   1:  PR[91,1] = PR[90,1] + -17.467;
   1:  PR[91,2] = PR[90,2] + 18.172;
   1:  PR[91,3] = PR[90,3] + 44.691;
   1:L PR[91] R[100]mm/sec CNT100;
   1:  PR[91,1] = PR[90,1] + -18.396;
   1:  PR[91,2] = PR[90,2] + 17.648;
   1:  PR[91,3] = PR[90,3] + 44.700;
   1:L PR[91] R[100]mm/sec CNT100;
   1:  PR[91,1] = PR[90,1] + -19.296;
   1:  PR[91,2] = PR[90,2] + 17.079;
   1:  PR[91,3] = PR[90,3] + 44.709;
   1:L PR[91] R[100]mm/sec CNT100;
   1:  PR[91,1] = PR[90,1] + -19.802;
   1:  PR[91,2] = PR[90,2] + 16.724;
   1:  PR[91,3] = PR[90,3] + 44.717;
   1:L PR[91] R[100]mm/sec CNT100;
   1:  PR[91,1] = PR[90,1] + -20.163;
   1:  PR[91,2] = PR[90,2] + 16.469;
   1:  PR[91,3] = PR[90,3] + 44.723;
   1:L PR[91] R[100]mm/sec CNT100;
   1:  PR[91,1] = PR[90,1] + -20.998;
   1:  PR[91,2] = PR[90,2] + 15.816;
   1:  PR[91,3] = PR[90,3] + 44.726;
   1:L PR[91] R[100]mm/sec CNT100;
   1:  PR[91,1] = PR[90,1] + -21.796;
   1:  PR[91,2] = PR[90,2] + 15.125;
   1:  PR[91,3] = PR[90,3] + 44.735;
   1:L PR[91] R[100]mm/sec CNT100;
   1:  PR[91,1] = PR[90,1] + -22.555;
   1:  PR[91,2] = PR[90,2] + 14.396;
   1:  PR[91,3] = PR[90,3] + 44.744;
   1:L PR[91] R[100]mm/sec CNT100;
   1:  PR[91,1] = PR[90,1] + -23.275;
   1:  PR[91,2] = PR[90,2] + 13.631;
   1:  PR[91,3] = PR[90,3] + 44.753;
   1:L PR[91] R[100]mm/sec CNT100;
   1:  PR[91,1] = PR[90,1] + -23.953;
   1:  PR[91,2] = PR[90,2] + 12.831;
   1:  PR[91,3] = PR[90,3] + 44.762;
   1:L PR[91] R[100]mm/sec CNT100;
   1:  PR[91,1] = PR[90,1] + -24.588;
   1:  PR[91,2] = PR[90,2] + 11.999;
   1:  PR[91,3] = PR[90,3] + 44.770;
   1:L PR[91] R[100]mm/sec CNT100;
   1:  PR[91,1] = PR[90,1] + -25.178;
   1:  PR[91,2] = PR[90,2] + 11.136;
   1:  PR[91,3] = PR[90,3] + 44.779;
   1:L PR[91] R[100]mm/sec CNT100;
   1:  PR[91,1] = PR[90,1] + -25.721;
   1:  PR[91,2] = PR[90,2] + 10.245;
   1:  PR[91,3] = PR[90,3] + 44.788;
   1:L PR[91] R[100]mm/sec CNT100;
   1:  PR[91,1] = PR[90,1] + -26.217;
   1:  PR[91,2] = PR[90,2] + 9.330;
   1:  PR[91,3] = PR[90,3] + 44.797;
   1:L PR[91] R[100]mm/sec CNT100;
   1:  PR[91,1] = PR[90,1] + -26.665;
   1:  PR[91,2] = PR[90,2] + 8.395;
   1:  PR[91,3] = PR[90,3] + 44.805;
   1:L PR[91] R[100]mm/sec CNT100;
   1:  PR[91,1] = PR[90,1] + -27.062;
   1:  PR[91,2] = PR[90,2] + 7.445;
   1:  PR[91,3] = PR[90,3] + 44.814;
   1:L PR[91] R[100]mm/sec CNT100;
   1:  PR[91,1] = PR[90,1] + -27.408;
   1:  PR[91,2] = PR[90,2] + 6.483;
   1:  PR[91,3] = PR[90,3] + 44.823;
   1:L PR[91] R[100]mm/sec CNT100;
   1:  PR[91,1] = PR[90,1] + -27.702;
   1:  PR[91,2] = PR[90,2] + 5.510;
   1:  PR[91,3] = PR[90,3] + 44.831;
   1:L PR[91] R[100]mm/sec CNT100;
   1:  PR[91,1] = PR[90,1] + -27.944;
   1:  PR[91,2] = PR[90,2] + 4.526;
   1:  PR[91,3] = PR[90,3] + 44.840;
   1:L PR[91] R[100]mm/sec CNT100;
   1:  PR[91,1] = PR[90,1] + -28.133;
   1:  PR[91,2] = PR[90,2] + 3.530;
   1:  PR[91,3] = PR[90,3] + 44.848;
   1:L PR[91] R[100]mm/sec CNT100;
   1:  PR[91,1] = PR[90,1] + -28.268;
   1:  PR[91,2] = PR[90,2] + 2.517;
   1:  PR[91,3] = PR[90,3] + 44.857;
   1:L PR[91] R[100]mm/sec CNT100;
   1:  PR[91,1] = PR[90,1] + -28.349;
   1:  PR[91,2] = PR[90,2] + 1.484;
   1:  PR[91,3] = PR[90,3] + 44.865;
   1:L PR[91] R[100]mm/sec CNT100;
   1:  PR[91,1] = PR[90,1] + -28.375;
   1:  PR[91,2] = PR[90,2] + 0.428;
   1:  PR[91,3] = PR[90,3] + 44.874;
   1:L PR[91] R[100]mm/sec CNT100;
   1:  PR[91,1] = PR[90,1] + -28.349;
   1:  PR[91,2] = PR[90,2] + -0.629;
   1:  PR[91,3] = PR[90,3] + 44.883;
   1:L PR[91] R[100]mm/sec CNT100;
   1:  PR[91,1] = PR[90,1] + -28.268;
   1:  PR[91,2] = PR[90,2] + -1.662;
   1:  PR[91,3] = PR[90,3] + 44.892;
   1:L PR[91] R[100]mm/sec CNT100;
   1:  PR[91,1] = PR[90,1] + -28.133;
   1:  PR[91,2] = PR[90,2] + -2.675;
   1:  PR[91,3] = PR[90,3] + 44.900;
   1:L PR[91] R[100]mm/sec CNT100;
   1:  PR[91,1] = PR[90,1] + -27.941;
   1:  PR[91,2] = PR[90,2] + -3.683;
   1:  PR[91,3] = PR[90,3] + 44.909;
   1:L PR[91] R[100]mm/sec CNT100;
   1:  PR[91,1] = PR[90,1] + -27.702;
   1:  PR[91,2] = PR[90,2] + -4.656;
   1:  PR[91,3] = PR[90,3] + 44.917;
   1:L PR[91] R[100]mm/sec CNT100;
   1:  PR[91,1] = PR[90,1] + -27.402;
   1:  PR[91,2] = PR[90,2] + -5.645;
   1:  PR[91,3] = PR[90,3] + 44.926;
   1:L PR[91] R[100]mm/sec CNT100;
   1:  PR[91,1] = PR[90,1] + -27.062;
   1:  PR[91,2] = PR[90,2] + -6.590;
   1:  PR[91,3] = PR[90,3] + 44.934;
   1:L PR[91] R[100]mm/sec CNT100;
   1:  PR[91,1] = PR[90,1] + -26.665;
   1:  PR[91,2] = PR[90,2] + -7.540;
   1:  PR[91,3] = PR[90,3] + 44.943;
   1:L PR[91] R[100]mm/sec CNT100;
   1:  PR[91,1] = PR[90,1] + -26.217;
   1:  PR[91,2] = PR[90,2] + -8.475;
   1:  PR[91,3] = PR[90,3] + 44.951;
   1:L PR[91] R[100]mm/sec CNT100;
   1:  PR[91,1] = PR[90,1] + -25.721;
   1:  PR[91,2] = PR[90,2] + -9.390;
   1:  PR[91,3] = PR[90,3] + 44.960;
   1:L PR[91] R[100]mm/sec CNT100;
   1:  PR[91,1] = PR[90,1] + -25.178;
   1:  PR[91,2] = PR[90,2] + -10.281;
   1:  PR[91,3] = PR[90,3] + 44.969;
   1:L PR[91] R[100]mm/sec CNT100;
   1:  PR[91,1] = PR[90,1] + -24.588;
   1:  PR[91,2] = PR[90,2] + -11.144;
   1:  PR[91,3] = PR[90,3] + 44.977;
   1:L PR[91] R[100]mm/sec CNT100;
   1:  PR[91,1] = PR[90,1] + -23.953;
   1:  PR[91,2] = PR[90,2] + -11.976;
   1:  PR[91,3] = PR[90,3] + 44.986;
   1:L PR[91] R[100]mm/sec CNT100;
   1:  PR[91,1] = PR[90,1] + -23.275;
   1:  PR[91,2] = PR[90,2] + -12.776;
   1:  PR[91,3] = PR[90,3] + 44.995;
   1:L PR[91] R[100]mm/sec CNT100;
   1:  PR[91,1] = PR[90,1] + -22.555;
   1:  PR[91,2] = PR[90,2] + -13.541;
   1:  PR[91,3] = PR[90,3] + 45.004;
   1:L PR[91] R[100]mm/sec CNT100;
   1:  PR[91,1] = PR[90,1] + -21.796;
   1:  PR[91,2] = PR[90,2] + -14.270;
   1:  PR[91,3] = PR[90,3] + 45.013;
   1:L PR[91] R[100]mm/sec CNT100;
   1:  PR[91,1] = PR[90,1] + -20.998;
   1:  PR[91,2] = PR[90,2] + -14.961;
   1:  PR[91,3] = PR[90,3] + 45.021;
   1:L PR[91] R[100]mm/sec CNT100;
   1:  PR[91,1] = PR[90,1] + -20.164;
   1:  PR[91,2] = PR[90,2] + -15.613;
   1:  PR[91,3] = PR[90,3] + 45.030;
   1:L PR[91] R[100]mm/sec CNT100;
   1:  PR[91,1] = PR[90,1] + -19.296;
   1:  PR[91,2] = PR[90,2] + -16.224;
   1:  PR[91,3] = PR[90,3] + 45.039;
   1:L PR[91] R[100]mm/sec CNT100;
   1:  PR[91,1] = PR[90,1] + -18.396;
   1:  PR[91,2] = PR[90,2] + -16.793;
   1:  PR[91,3] = PR[90,3] + 45.048;
   1:L PR[91] R[100]mm/sec CNT100;
   1:  PR[91,1] = PR[90,1] + -17.921;
   1:  PR[91,2] = PR[90,2] + -17.062;
   1:  PR[91,3] = PR[90,3] + 45.057;
   1:L PR[91] R[100]mm/sec CNT100;
   1:  PR[91,1] = PR[90,1] + -17.468;
   1:  PR[91,2] = PR[90,2] + -17.317;
   1:  PR[91,3] = PR[90,3] + 45.061;
   1:L PR[91] R[100]mm/sec CNT100;
   1:  PR[91,1] = PR[90,1] + -16.511;
   1:  PR[91,2] = PR[90,2] + -17.796;
   1:  PR[91,3] = PR[90,3] + 45.066;
   1:L PR[91] R[100]mm/sec CNT100;
   1:  PR[91,1] = PR[90,1] + -15.531;
   1:  PR[91,2] = PR[90,2] + -18.227;
   1:  PR[91,3] = PR[90,3] + 45.075;
   1:L PR[91] R[100]mm/sec CNT100;
   1:  PR[91,1] = PR[90,1] + -14.528;
   1:  PR[91,2] = PR[90,2] + -18.610;
   1:  PR[91,3] = PR[90,3] + 45.084;
   1:L PR[91] R[100]mm/sec CNT100;
   1:  PR[91,1] = PR[90,1] + -13.506;
   1:  PR[91,2] = PR[90,2] + -18.943;
   1:  PR[91,3] = PR[90,3] + 45.093;
   1:L PR[91] R[100]mm/sec CNT100;
   1:  PR[91,1] = PR[90,1] + -12.468;
   1:  PR[91,2] = PR[90,2] + -19.224;
   1:  PR[91,3] = PR[90,3] + 45.102;
   1:L PR[91] R[100]mm/sec CNT100;
   1:  PR[91,1] = PR[90,1] + -11.415;
   1:  PR[91,2] = PR[90,2] + -19.455;
   1:  PR[91,3] = PR[90,3] + 45.111;
   1:L PR[91] R[100]mm/sec CNT100;
   1:  PR[91,1] = PR[90,1] + -10.351;
   1:  PR[91,2] = PR[90,2] + -19.632;
   1:  PR[91,3] = PR[90,3] + 45.120;
   1:L PR[91] R[100]mm/sec CNT100;
   1:  PR[91,1] = PR[90,1] + -9.279;
   1:  PR[91,2] = PR[90,2] + -19.757;
   1:  PR[91,3] = PR[90,3] + 45.129;
   1:L PR[91] R[100]mm/sec CNT100;
   1:  PR[91,1] = PR[90,1] + -8.201;
   1:  PR[91,2] = PR[90,2] + -19.828;
   1:  PR[91,3] = PR[90,3] + 45.138;
   1:L PR[91] R[100]mm/sec CNT100;
   1:  PR[91,1] = PR[90,1] + -7.114;
   1:  PR[91,2] = PR[90,2] + -19.846;
   1:  PR[91,3] = PR[90,3] + 45.147;
   1:L PR[91] R[100]mm/sec CNT100;
   1:  PR[91,1] = PR[90,1] + -6.036;
   1:  PR[91,2] = PR[90,2] + -19.811;
   1:  PR[91,3] = PR[90,3] + 45.156;
   1:L PR[91] R[100]mm/sec CNT100;
   1:  PR[91,1] = PR[90,1] + -4.956;
   1:  PR[91,2] = PR[90,2] + -19.721;
   1:  PR[91,3] = PR[90,3] + 45.165;
   1:L PR[91] R[100]mm/sec CNT100;
   1:  PR[91,1] = PR[90,1] + -3.881;
   1:  PR[91,2] = PR[90,2] + -19.578;
   1:  PR[91,3] = PR[90,3] + 45.174;
   1:L PR[91] R[100]mm/sec CNT100;
   1:  PR[91,1] = PR[90,1] + -2.816;
   1:  PR[91,2] = PR[90,2] + -19.380;
   1:  PR[91,3] = PR[90,3] + 45.183;
   1:L PR[91] R[100]mm/sec CNT100;
   1:  PR[91,1] = PR[90,1] + -1.760;
   1:  PR[91,2] = PR[90,2] + -19.128;
   1:  PR[91,3] = PR[90,3] + 45.192;
   1:L PR[91] R[100]mm/sec CNT100;
   1:  PR[91,1] = PR[90,1] + -0.975;
   1:  PR[91,2] = PR[90,2] + -18.899;
   1:  PR[91,3] = PR[90,3] + 45.201;
   1:L PR[91] R[100]mm/sec CNT100;
   1:  PR[91,1] = PR[90,1] + -0.725;
   1:  PR[91,2] = PR[90,2] + -18.841;
   1:  PR[91,3] = PR[90,3] + 45.208;
   1:L PR[91] R[100]mm/sec CNT100;
   1:  PR[91,1] = PR[90,1] + -0.517;
   1:  PR[91,2] = PR[90,2] + -18.799;
   1:  PR[91,3] = PR[90,3] + 45.210;
   1:L PR[91] R[100]mm/sec CNT100;
   1:  PR[91,1] = PR[90,1] + -0.033;
   1:  PR[91,2] = PR[90,2] + -18.773;
   1:  PR[91,3] = PR[90,3] + 45.212;
   1:L PR[91] R[100]mm/sec CNT100;
   1:  PR[91,1] = PR[90,1] + 0.455;
   1:  PR[91,2] = PR[90,2] + -18.828;
   1:  PR[91,3] = PR[90,3] + 45.216;
   1:L PR[91] R[100]mm/sec CNT100;
   1:  PR[91] = PR[90];
   1:  PR[91,1] = PR[90,1] + 0.991;
   1:  PR[91,2] = PR[90,2] + -19.358;
   1:  PR[91,3] = PR[90,3] + 46.550;
   1:L PR[91] R[100]mm/sec CNT100;
   1:  PR[91,1] = PR[90,1] + 2.061;
   1:  PR[91,2] = PR[90,2] + -19.613;
   1:  PR[91,3] = PR[90,3] + 45.224;
   1:L PR[91] R[100]mm/sec CNT100;
   1:  PR[91,1] = PR[90,1] + 3.136;
   1:  PR[91,2] = PR[90,2] + -19.812;
   1:  PR[91,3] = PR[90,3] + 45.233;
   1:L PR[91] R[100]mm/sec CNT100;
   1:  PR[91,1] = PR[90,1] + 4.218;
   1:  PR[91,2] = PR[90,2] + -19.956;
   1:  PR[91,3] = PR[90,3] + 45.243;
   1:L PR[91] R[100]mm/sec CNT100;
   1:  PR[91,1] = PR[90,1] + 5.307;
   1:  PR[91,2] = PR[90,2] + -20.046;
   1:  PR[91,3] = PR[90,3] + 45.252;
   1:L PR[91] R[100]mm/sec CNT100;
   1:  PR[91,1] = PR[90,1] + 6.398;
   1:  PR[91,2] = PR[90,2] + -20.080;
   1:  PR[91,3] = PR[90,3] + 45.261;
   1:L PR[91] R[100]mm/sec CNT100;
   1:  PR[91,1] = PR[90,1] + 7.490;
   1:  PR[91,2] = PR[90,2] + -20.060;
   1:  PR[91,3] = PR[90,3] + 45.270;
   1:L PR[91] R[100]mm/sec CNT100;
   1:  PR[91,1] = PR[90,1] + 8.578;
   1:  PR[91,2] = PR[90,2] + -19.986;
   1:  PR[91,3] = PR[90,3] + 45.279;
   1:L PR[91] R[100]mm/sec CNT100;
   1:  PR[91,1] = PR[90,1] + 9.660;
   1:  PR[91,2] = PR[90,2] + -19.857;
   1:  PR[91,3] = PR[90,3] + 45.288;
   1:L PR[91] R[100]mm/sec CNT100;
   1:  PR[91,1] = PR[90,1] + 10.734;
   1:  PR[91,2] = PR[90,2] + -19.675;
   1:  PR[91,3] = PR[90,3] + 45.298;
   1:L PR[91] R[100]mm/sec CNT100;
   1:  PR[91,1] = PR[90,1] + 11.795;
   1:  PR[91,2] = PR[90,2] + -19.439;
   1:  PR[91,3] = PR[90,3] + 45.307;
   1:L PR[91] R[100]mm/sec CNT100;
   1:  PR[91,1] = PR[90,1] + 12.843;
   1:  PR[91,2] = PR[90,2] + -19.151;
   1:  PR[91,3] = PR[90,3] + 45.316;
   1:L PR[91] R[100]mm/sec CNT100;
   1:  PR[91,1] = PR[90,1] + 13.873;
   1:  PR[91,2] = PR[90,2] + -18.812;
   1:  PR[91,3] = PR[90,3] + 45.325;
   1:L PR[91] R[100]mm/sec CNT100;
   1:  PR[91,1] = PR[90,1] + 14.883;
   1:  PR[91,2] = PR[90,2] + -18.423;
   1:  PR[91,3] = PR[90,3] + 45.334;
   1:L PR[91] R[100]mm/sec CNT100;
   1:  PR[91,1] = PR[90,1] + 15.871;
   1:  PR[91,2] = PR[90,2] + -17.985;
   1:  PR[91,3] = PR[90,3] + 45.343;
   1:L PR[91] R[100]mm/sec CNT100;
   1:  PR[91,1] = PR[90,1] + 16.834;
   1:  PR[91,2] = PR[90,2] + -17.499;
   1:  PR[91,3] = PR[90,3] + 45.352;
   1:L PR[91] R[100]mm/sec CNT100;
   1:  PR[91,1] = PR[90,1] + 17.777;
   1:  PR[91,2] = PR[90,2] + -16.964;
   1:  PR[91,3] = PR[90,3] + 45.361;
   1:L PR[91] R[100]mm/sec CNT100;
   1:  PR[91,1] = PR[90,1] + 18.675;
   1:  PR[91,2] = PR[90,2] + -16.394;
   1:  PR[91,3] = PR[90,3] + 45.371;
   1:L PR[91] R[100]mm/sec CNT100;
   1:  PR[91,1] = PR[90,1] + 19.548;
   1:  PR[91,2] = PR[90,2] + -15.776;
   1:  PR[91,3] = PR[90,3] + 45.379;
   1:L PR[91] R[100]mm/sec CNT100;
   1:  PR[91,1] = PR[90,1] + 20.387;
   1:  PR[91,2] = PR[90,2] + -15.117;
   1:  PR[91,3] = PR[90,3] + 45.388;
   1:L PR[91] R[100]mm/sec CNT100;
   1:  PR[91,1] = PR[90,1] + 21.190;
   1:  PR[91,2] = PR[90,2] + -14.418;
   1:  PR[91,3] = PR[90,3] + 45.397;
   1:L PR[91] R[100]mm/sec CNT100;
   1:  PR[91,1] = PR[90,1] + 21.955;
   1:  PR[91,2] = PR[90,2] + -13.681;
   1:  PR[91,3] = PR[90,3] + 45.406;
   1:L PR[91] R[100]mm/sec CNT100;
   1:  PR[91,1] = PR[90,1] + 22.679;
   1:  PR[91,2] = PR[90,2] + -12.906;
   1:  PR[91,3] = PR[90,3] + 45.415;
   1:L PR[91] R[100]mm/sec CNT100;
   1:  PR[91,1] = PR[90,1] + 23.361;
   1:  PR[91,2] = PR[90,2] + -12.097;
   1:  PR[91,3] = PR[90,3] + 45.424;
   1:L PR[91] R[100]mm/sec CNT100;
   1:  PR[91,1] = PR[90,1] + 24.000;
   1:  PR[91,2] = PR[90,2] + -11.255;
   1:  PR[91,3] = PR[90,3] + 45.433;
   1:L PR[91] R[100]mm/sec CNT100;
   1:  PR[91,1] = PR[90,1] + 24.594;
   1:  PR[91,2] = PR[90,2] + -10.383;
   1:  PR[91,3] = PR[90,3] + 45.442;
   1:L PR[91] R[100]mm/sec CNT100;
   1:  PR[91,1] = PR[90,1] + 25.141;
   1:  PR[91,2] = PR[90,2] + -9.484;
   1:  PR[91,3] = PR[90,3] + 45.451;
   1:L PR[91] R[100]mm/sec CNT100;
   1:  PR[91,1] = PR[90,1] + 25.640;
   1:  PR[91,2] = PR[90,2] + -8.563;
   1:  PR[91,3] = PR[90,3] + 45.460;
   1:L PR[91] R[100]mm/sec CNT100;
   1:  PR[91,1] = PR[90,1] + 26.091;
   1:  PR[91,2] = PR[90,2] + -7.622;
   1:  PR[91,3] = PR[90,3] + 45.469;
   1:L PR[91] R[100]mm/sec CNT100;
   1:  PR[91,1] = PR[90,1] + 26.490;
   1:  PR[91,2] = PR[90,2] + -6.665;
   1:  PR[91,3] = PR[90,3] + 45.477;
   1:L PR[91] R[100]mm/sec CNT100;
   1:  PR[91,1] = PR[90,1] + 26.838;
   1:  PR[91,2] = PR[90,2] + -5.696;
   1:  PR[91,3] = PR[90,3] + 45.486;
   1:L PR[91] R[100]mm/sec CNT100;
   1:  PR[91,1] = PR[90,1] + 27.134;
   1:  PR[91,2] = PR[90,2] + -4.714;
   1:  PR[91,3] = PR[90,3] + 45.495;
   1:L PR[91] R[100]mm/sec CNT100;
   1:  PR[91,1] = PR[90,1] + 27.377;
   1:  PR[91,2] = PR[90,2] + -3.719;
   1:  PR[91,3] = PR[90,3] + 45.503;
   1:L PR[91] R[100]mm/sec CNT100;
   1:  PR[91,1] = PR[90,1] + 27.566;
   1:  PR[91,2] = PR[90,2] + -2.710;
   1:  PR[91,3] = PR[90,3] + 45.512;
   1:L PR[91] R[100]mm/sec CNT100;
   1:  PR[91,1] = PR[90,1] + 27.702;
   1:  PR[91,2] = PR[90,2] + -1.683;
   1:  PR[91,3] = PR[90,3] + 45.521;
   1:L PR[91] R[100]mm/sec CNT100;
   1:  PR[91,1] = PR[90,1] + 27.784;
   1:  PR[91,2] = PR[90,2] + -0.638;
   1:  PR[91,3] = PR[90,3] + 45.529;
   1:L PR[91] R[100]mm/sec CNT100;
   1:  PR[91,1] = PR[90,1] + 27.811;
   1:  PR[91,2] = PR[90,2] + 0.428;
   1:  PR[91,3] = PR[90,3] + 45.538;
   1:L PR[91] R[100]mm/sec CNT100;
   1:  PR[91,1] = PR[90,1] + 27.784;
   1:  PR[91,2] = PR[90,2] + 1.493;
   1:  PR[91,3] = PR[90,3] + 45.547;
   1:L PR[91] R[100]mm/sec CNT100;
   1:  PR[91,1] = PR[90,1] + 27.702;
   1:  PR[91,2] = PR[90,2] + 2.538;
   1:  PR[91,3] = PR[90,3] + 45.556;
   1:L PR[91] R[100]mm/sec CNT100;
   1:  PR[91,1] = PR[90,1] + 27.566;
   1:  PR[91,2] = PR[90,2] + 3.565;
   1:  PR[91,3] = PR[90,3] + 45.565;
   1:L PR[91] R[100]mm/sec CNT100;
   1:  PR[91,1] = PR[90,1] + 27.377;
   1:  PR[91,2] = PR[90,2] + 4.574;
   1:  PR[91,3] = PR[90,3] + 45.574;
   1:L PR[91] R[100]mm/sec CNT100;
   1:  PR[91,1] = PR[90,1] + 27.134;
   1:  PR[91,2] = PR[90,2] + 5.569;
   1:  PR[91,3] = PR[90,3] + 45.582;
   1:L PR[91] R[100]mm/sec CNT100;
   1:  PR[91,1] = PR[90,1] + 26.838;
   1:  PR[91,2] = PR[90,2] + 6.551;
   1:  PR[91,3] = PR[90,3] + 45.591;
   1:L PR[91] R[100]mm/sec CNT100;
   1:  PR[91,1] = PR[90,1] + 26.490;
   1:  PR[91,2] = PR[90,2] + 7.520;
   1:  PR[91,3] = PR[90,3] + 45.599;
   1:L PR[91] R[100]mm/sec CNT100;
   1:  PR[91,1] = PR[90,1] + 26.091;
   1:  PR[91,2] = PR[90,2] + 8.477;
   1:  PR[91,3] = PR[90,3] + 45.608;
   1:L PR[91] R[100]mm/sec CNT100;
   1:  PR[91,1] = PR[90,1] + 25.641;
   1:  PR[91,2] = PR[90,2] + 9.417;
   1:  PR[91,3] = PR[90,3] + 45.617;
   1:L PR[91] R[100]mm/sec CNT100;
   1:  PR[91,1] = PR[90,1] + 25.141;
   1:  PR[91,2] = PR[90,2] + 10.339;
   1:  PR[91,3] = PR[90,3] + 45.626;
   1:L PR[91] R[100]mm/sec CNT100;
   1:  PR[91,1] = PR[90,1] + 24.594;
   1:  PR[91,2] = PR[90,2] + 11.238;
   1:  PR[91,3] = PR[90,3] + 45.634;
   1:L PR[91] R[100]mm/sec CNT100;
   1:  PR[91,1] = PR[90,1] + 24.000;
   1:  PR[91,2] = PR[90,2] + 12.110;
   1:  PR[91,3] = PR[90,3] + 45.643;
   1:L PR[91] R[100]mm/sec CNT100;
   1:  PR[91,1] = PR[90,1] + 23.362;
   1:  PR[91,2] = PR[90,2] + 12.952;
   1:  PR[91,3] = PR[90,3] + 45.652;
   1:L PR[91] R[100]mm/sec CNT100;
   1:  PR[91,1] = PR[90,1] + 22.679;
   1:  PR[91,2] = PR[90,2] + 13.761;
   1:  PR[91,3] = PR[90,3] + 45.661;
   1:L PR[91] R[100]mm/sec CNT100;
   1:  PR[91,1] = PR[90,1] + 21.955;
   1:  PR[91,2] = PR[90,2] + 14.535;
   1:  PR[91,3] = PR[90,3] + 45.670;
   1:L PR[91] R[100]mm/sec CNT100;
   1:  PR[91,1] = PR[90,1] + 21.191;
   1:  PR[91,2] = PR[90,2] + 15.273;
   1:  PR[91,3] = PR[90,3] + 45.679;
   1:L PR[91] R[100]mm/sec CNT100;
   1:  PR[91,1] = PR[90,1] + 20.388;
   1:  PR[91,2] = PR[90,2] + 15.972;
   1:  PR[91,3] = PR[90,3] + 45.688;
   1:L PR[91] R[100]mm/sec CNT100;
   1:  PR[91,1] = PR[90,1] + 19.549;
   1:  PR[91,2] = PR[90,2] + 16.631;
   1:  PR[91,3] = PR[90,3] + 45.697;
   1:L PR[91] R[100]mm/sec CNT100;
   1:  PR[91,1] = PR[90,1] + 18.676;
   1:  PR[91,2] = PR[90,2] + 17.248;
   1:  PR[91,3] = PR[90,3] + 45.706;
   1:L PR[91] R[100]mm/sec CNT100;
   1:  PR[91,1] = PR[90,1] + 17.771;
   1:  PR[91,2] = PR[90,2] + 17.823;
   1:  PR[91,3] = PR[90,3] + 45.715;
   1:L PR[91] R[100]mm/sec CNT100;
   1:  PR[91,1] = PR[90,1] + 16.835;
   1:  PR[91,2] = PR[90,2] + 18.354;
   1:  PR[91,3] = PR[90,3] + 45.724;
   1:L PR[91] R[100]mm/sec CNT100;
   1:  PR[91,1] = PR[90,1] + 15.872;
   1:  PR[91,2] = PR[90,2] + 18.839;
   1:  PR[91,3] = PR[90,3] + 45.733;
   1:L PR[91] R[100]mm/sec CNT100;
   1:  PR[91,1] = PR[90,1] + 14.885;
   1:  PR[91,2] = PR[90,2] + 19.277;
   1:  PR[91,3] = PR[90,3] + 45.742;
   1:L PR[91] R[100]mm/sec CNT100;
   1:  PR[91,1] = PR[90,1] + 13.874;
   1:  PR[91,2] = PR[90,2] + 19.667;
   1:  PR[91,3] = PR[90,3] + 45.751;
   1:L PR[91] R[100]mm/sec CNT100;
   1:  PR[91,1] = PR[90,1] + 12.844;
   1:  PR[91,2] = PR[90,2] + 20.006;
   1:  PR[91,3] = PR[90,3] + 45.760;
   1:L PR[91] R[100]mm/sec CNT100;
   1:  PR[91,1] = PR[90,1] + 11.797;
   1:  PR[91,2] = PR[90,2] + 20.294;
   1:  PR[91,3] = PR[90,3] + 45.769;
   1:L PR[91] R[100]mm/sec CNT100;
   1:  PR[91,1] = PR[90,1] + 10.735;
   1:  PR[91,2] = PR[90,2] + 20.529;
   1:  PR[91,3] = PR[90,3] + 45.778;
   1:L PR[91] R[100]mm/sec CNT100;
   1:  PR[91,1] = PR[90,1] + 9.662;
   1:  PR[91,2] = PR[90,2] + 20.712;
   1:  PR[91,3] = PR[90,3] + 45.787;
   1:L PR[91] R[100]mm/sec CNT100;
   1:  PR[91,1] = PR[90,1] + 8.579;
   1:  PR[91,2] = PR[90,2] + 20.841;
   1:  PR[91,3] = PR[90,3] + 45.797;
   1:L PR[91] R[100]mm/sec CNT100;
   1:  PR[91,1] = PR[90,1] + 7.491;
   1:  PR[91,2] = PR[90,2] + 20.915;
   1:  PR[91,3] = PR[90,3] + 45.806;
   1:L PR[91] R[100]mm/sec CNT100;
   1:  PR[91,1] = PR[90,1] + 6.400;
   1:  PR[91,2] = PR[90,2] + 20.935;
   1:  PR[91,3] = PR[90,3] + 45.815;
   1:L PR[91] R[100]mm/sec CNT100;
   1:  PR[91,1] = PR[90,1] + 5.309;
   1:  PR[91,2] = PR[90,2] + 20.901;
   1:  PR[91,3] = PR[90,3] + 45.824;
   1:L PR[91] R[100]mm/sec CNT100;
   1:  PR[91,1] = PR[90,1] + 4.220;
   1:  PR[91,2] = PR[90,2] + 20.812;
   1:  PR[91,3] = PR[90,3] + 45.833;
   1:L PR[91] R[100]mm/sec CNT100;
   1:  PR[91,1] = PR[90,1] + 3.137;
   1:  PR[91,2] = PR[90,2] + 20.667;
   1:  PR[91,3] = PR[90,3] + 45.842;
   1:L PR[91] R[100]mm/sec CNT100;
   1:  PR[91,1] = PR[90,1] + 2.063;
   1:  PR[91,2] = PR[90,2] + 20.469;
   1:  PR[91,3] = PR[90,3] + 45.852;
   1:L PR[91] R[100]mm/sec CNT100;
   1:  PR[91,1] = PR[90,1] + 0.994;
   1:  PR[91,2] = PR[90,2] + 20.214;
   1:  PR[91,3] = PR[90,3] + 45.861;
   1:L PR[91] R[100]mm/sec CNT100;
   1:  PR[91,1] = PR[90,1] + 0.516;
   1:  PR[91,2] = PR[90,2] + 20.083;
   1:  PR[91,3] = PR[90,3] + 45.870;
   1:L PR[91] R[100]mm/sec CNT100;
   1:  PR[91,1] = PR[90,1] + 0.038;
   1:  PR[91,2] = PR[90,2] + 20.019;
   1:  PR[91,3] = PR[90,3] + 45.874;
   1:L PR[91] R[100]mm/sec CNT100;
   1:  PR[91,1] = PR[90,1] + -0.452;
   1:  PR[91,2] = PR[90,2] + 20.033;
   1:  PR[91,3] = PR[90,3] + 45.878;
   1:L PR[91] R[100]mm/sec CNT100;
   1:  PR[91,1] = PR[90,1] + -0.908;
   1:  PR[91,2] = PR[90,2] + 20.122;
   1:  PR[91,3] = PR[90,3] + 45.882;
   1:L PR[91] R[100]mm/sec CNT100;
   1:  PR[91,1] = PR[90,1] + -1.233;
   1:  PR[91,2] = PR[90,2] + 20.215;
   1:  PR[91,3] = PR[90,3] + 45.886;
   1:L PR[91] R[100]mm/sec CNT100;
   1:  PR[91,1] = PR[90,1] + -2.299;
   1:  PR[91,2] = PR[90,2] + 20.468;
   1:  PR[91,3] = PR[90,3] + 45.889;
   1:L PR[91] R[100]mm/sec CNT100;
   1:  PR[91,1] = PR[90,1] + -3.373;
   1:  PR[91,2] = PR[90,2] + 20.667;
   1:  PR[91,3] = PR[90,3] + 45.898;
   1:L PR[91] R[100]mm/sec CNT100;
   1:  PR[91,1] = PR[90,1] + -4.456;
   1:  PR[91,2] = PR[90,2] + 20.811;
   1:  PR[91,3] = PR[90,3] + 45.908;
   1:L PR[91] R[100]mm/sec CNT100;
   1:  PR[91,1] = PR[90,1] + -5.545;
   1:  PR[91,2] = PR[90,2] + 20.901;
   1:  PR[91,3] = PR[90,3] + 45.917;
   1:L PR[91] R[100]mm/sec CNT100;
   1:  PR[91,1] = PR[90,1] + -6.636;
   1:  PR[91,2] = PR[90,2] + 20.935;
   1:  PR[91,3] = PR[90,3] + 45.926;
   1:L PR[91] R[100]mm/sec CNT100;
   1:  PR[91,1] = PR[90,1] + -7.728;
   1:  PR[91,2] = PR[90,2] + 20.915;
   1:  PR[91,3] = PR[90,3] + 45.935;
   1:L PR[91] R[100]mm/sec CNT100;
   1:  PR[91,1] = PR[90,1] + -8.816;
   1:  PR[91,2] = PR[90,2] + 20.841;
   1:  PR[91,3] = PR[90,3] + 45.944;
   1:L PR[91] R[100]mm/sec CNT100;
   1:  PR[91,1] = PR[90,1] + -9.898;
   1:  PR[91,2] = PR[90,2] + 20.712;
   1:  PR[91,3] = PR[90,3] + 45.953;
   1:L PR[91] R[100]mm/sec CNT100;
   1:  PR[91,1] = PR[90,1] + -10.972;
   1:  PR[91,2] = PR[90,2] + 20.530;
   1:  PR[91,3] = PR[90,3] + 45.963;
   1:L PR[91] R[100]mm/sec CNT100;
   1:  PR[91,1] = PR[90,1] + -12.034;
   1:  PR[91,2] = PR[90,2] + 20.294;
   1:  PR[91,3] = PR[90,3] + 45.972;
   1:L PR[91] R[100]mm/sec CNT100;
   1:  PR[91,1] = PR[90,1] + -13.081;
   1:  PR[91,2] = PR[90,2] + 20.007;
   1:  PR[91,3] = PR[90,3] + 45.981;
   1:L PR[91] R[100]mm/sec CNT100;
   1:  PR[91,1] = PR[90,1] + -14.111;
   1:  PR[91,2] = PR[90,2] + 19.668;
   1:  PR[91,3] = PR[90,3] + 45.990;
   1:L PR[91] R[100]mm/sec CNT100;
   1:  PR[91,1] = PR[90,1] + -15.121;
   1:  PR[91,2] = PR[90,2] + 19.279;
   1:  PR[91,3] = PR[90,3] + 45.999;
   1:L PR[91] R[100]mm/sec CNT100;
   1:  PR[91,1] = PR[90,1] + -16.109;
   1:  PR[91,2] = PR[90,2] + 18.840;
   1:  PR[91,3] = PR[90,3] + 46.008;
   1:L PR[91] R[100]mm/sec CNT100;
   1:  PR[91,1] = PR[90,1] + -17.072;
   1:  PR[91,2] = PR[90,2] + 18.354;
   1:  PR[91,3] = PR[90,3] + 46.017;
   1:L PR[91] R[100]mm/sec CNT100;
   1:  PR[91,1] = PR[90,1] + -18.015;
   1:  PR[91,2] = PR[90,2] + 17.818;
   1:  PR[91,3] = PR[90,3] + 46.026;
   1:L PR[91] R[100]mm/sec CNT100;
   1:  PR[91,1] = PR[90,1] + -18.914;
   1:  PR[91,2] = PR[90,2] + 17.247;
   1:  PR[91,3] = PR[90,3] + 46.036;
   1:L PR[91] R[100]mm/sec CNT100;
   1:  PR[91,1] = PR[90,1] + -19.787;
   1:  PR[91,2] = PR[90,2] + 16.630;
   1:  PR[91,3] = PR[90,3] + 46.044;
   1:L PR[91] R[100]mm/sec CNT100;
   1:  PR[91,1] = PR[90,1] + -20.626;
   1:  PR[91,2] = PR[90,2] + 15.971;
   1:  PR[91,3] = PR[90,3] + 46.053;
   1:L PR[91] R[100]mm/sec CNT100;
   1:  PR[91,1] = PR[90,1] + -21.429;
   1:  PR[91,2] = PR[90,2] + 15.272;
   1:  PR[91,3] = PR[90,3] + 46.062;
   1:L PR[91] R[100]mm/sec CNT100;
   1:  PR[91,1] = PR[90,1] + -22.193;
   1:  PR[91,2] = PR[90,2] + 14.536;
   1:  PR[91,3] = PR[90,3] + 46.071;
   1:L PR[91] R[100]mm/sec CNT100;
   1:  PR[91,1] = PR[90,1] + -22.918;
   1:  PR[91,2] = PR[90,2] + 13.763;
   1:  PR[91,3] = PR[90,3] + 46.080;
   1:L PR[91] R[100]mm/sec CNT100;
   1:  PR[91,1] = PR[90,1] + -23.600;
   1:  PR[91,2] = PR[90,2] + 12.955;
   1:  PR[91,3] = PR[90,3] + 46.089;
   1:L PR[91] R[100]mm/sec CNT100;
   1:  PR[91,1] = PR[90,1] + -24.239;
   1:  PR[91,2] = PR[90,2] + 12.115;
   1:  PR[91,3] = PR[90,3] + 46.098;
   1:L PR[91] R[100]mm/sec CNT100;
   1:  PR[91,1] = PR[90,1] + -24.832;
   1:  PR[91,2] = PR[90,2] + 11.243;
   1:  PR[91,3] = PR[90,3] + 46.107;
   1:L PR[91] R[100]mm/sec CNT100;
   1:  PR[91,1] = PR[90,1] + -25.379;
   1:  PR[91,2] = PR[90,2] + 10.344;
   1:  PR[91,3] = PR[90,3] + 46.116;
   1:L PR[91] R[100]mm/sec CNT100;
   1:  PR[91,1] = PR[90,1] + -25.879;
   1:  PR[91,2] = PR[90,2] + 9.420;
   1:  PR[91,3] = PR[90,3] + 46.125;
   1:L PR[91] R[100]mm/sec CNT100;
   1:  PR[91,1] = PR[90,1] + -26.329;
   1:  PR[91,2] = PR[90,2] + 8.476;
   1:  PR[91,3] = PR[90,3] + 46.134;
   1:L PR[91] R[100]mm/sec CNT100;
   1:  PR[91,1] = PR[90,1] + -26.728;
   1:  PR[91,2] = PR[90,2] + 7.516;
   1:  PR[91,3] = PR[90,3] + 46.142;
   1:L PR[91] R[100]mm/sec CNT100;
   1:  PR[91,1] = PR[90,1] + -27.077;
   1:  PR[91,2] = PR[90,2] + 6.544;
   1:  PR[91,3] = PR[90,3] + 46.151;
   1:L PR[91] R[100]mm/sec CNT100;
   1:  PR[91,1] = PR[90,1] + -27.373;
   1:  PR[91,2] = PR[90,2] + 5.560;
   1:  PR[91,3] = PR[90,3] + 46.160;
   1:L PR[91] R[100]mm/sec CNT100;
   1:  PR[91,1] = PR[90,1] + -27.615;
   1:  PR[91,2] = PR[90,2] + 4.566;
   1:  PR[91,3] = PR[90,3] + 46.168;
   1:L PR[91] R[100]mm/sec CNT100;
   1:  PR[91,1] = PR[90,1] + -27.805;
   1:  PR[91,2] = PR[90,2] + 3.558;
   1:  PR[91,3] = PR[90,3] + 46.177;
   1:L PR[91] R[100]mm/sec CNT100;
   1:  PR[91,1] = PR[90,1] + -27.941;
   1:  PR[91,2] = PR[90,2] + 2.535;
   1:  PR[91,3] = PR[90,3] + 46.186;
   1:L PR[91] R[100]mm/sec CNT100;
   1:  PR[91,1] = PR[90,1] + -28.022;
   1:  PR[91,2] = PR[90,2] + 1.492;
   1:  PR[91,3] = PR[90,3] + 46.194;
   1:L PR[91] R[100]mm/sec CNT100;
   1:  PR[91,1] = PR[90,1] + -28.050;
   1:  PR[91,2] = PR[90,2] + 0.428;
   1:  PR[91,3] = PR[90,3] + 46.203;
   1:L PR[91] R[100]mm/sec CNT100;
   1:  PR[91,1] = PR[90,1] + -28.022;
   1:  PR[91,2] = PR[90,2] + -0.637;
   1:  PR[91,3] = PR[90,3] + 46.212;
   1:L PR[91] R[100]mm/sec CNT100;
   1:  PR[91,1] = PR[90,1] + -27.941;
   1:  PR[91,2] = PR[90,2] + -1.680;
   1:  PR[91,3] = PR[90,3] + 46.221;
   1:L PR[91] R[100]mm/sec CNT100;
   1:  PR[91,1] = PR[90,1] + -27.805;
   1:  PR[91,2] = PR[90,2] + -2.703;
   1:  PR[91,3] = PR[90,3] + 46.230;
   1:L PR[91] R[100]mm/sec CNT100;
   1:  PR[91,1] = PR[90,1] + -27.615;
   1:  PR[91,2] = PR[90,2] + -3.711;
   1:  PR[91,3] = PR[90,3] + 46.239;
   1:L PR[91] R[100]mm/sec CNT100;
   1:  PR[91,1] = PR[90,1] + -27.373;
   1:  PR[91,2] = PR[90,2] + -4.705;
   1:  PR[91,3] = PR[90,3] + 46.247;
   1:L PR[91] R[100]mm/sec CNT100;
   1:  PR[91,1] = PR[90,1] + -27.077;
   1:  PR[91,2] = PR[90,2] + -5.689;
   1:  PR[91,3] = PR[90,3] + 46.256;
   1:L PR[91] R[100]mm/sec CNT100;
   1:  PR[91,1] = PR[90,1] + -26.728;
   1:  PR[91,2] = PR[90,2] + -6.661;
   1:  PR[91,3] = PR[90,3] + 46.264;
   1:L PR[91] R[100]mm/sec CNT100;
   1:  PR[91,1] = PR[90,1] + -26.329;
   1:  PR[91,2] = PR[90,2] + -7.621;
   1:  PR[91,3] = PR[90,3] + 46.273;
   1:L PR[91] R[100]mm/sec CNT100;
   1:  PR[91,1] = PR[90,1] + -25.878;
   1:  PR[91,2] = PR[90,2] + -8.565;
   1:  PR[91,3] = PR[90,3] + 46.282;
   1:L PR[91] R[100]mm/sec CNT100;
   1:  PR[91,1] = PR[90,1] + -25.379;
   1:  PR[91,2] = PR[90,2] + -9.489;
   1:  PR[91,3] = PR[90,3] + 46.291;
   1:L PR[91] R[100]mm/sec CNT100;
   1:  PR[91,1] = PR[90,1] + -24.832;
   1:  PR[91,2] = PR[90,2] + -10.388;
   1:  PR[91,3] = PR[90,3] + 46.299;
   1:L PR[91] R[100]mm/sec CNT100;
   1:  PR[91,1] = PR[90,1] + -24.239;
   1:  PR[91,2] = PR[90,2] + -11.260;
   1:  PR[91,3] = PR[90,3] + 46.308;
   1:L PR[91] R[100]mm/sec CNT100;
   1:  PR[91,1] = PR[90,1] + -23.600;
   1:  PR[91,2] = PR[90,2] + -12.100;
   1:  PR[91,3] = PR[90,3] + 46.317;
   1:L PR[91] R[100]mm/sec CNT100;
   1:  PR[91,1] = PR[90,1] + -22.917;
   1:  PR[91,2] = PR[90,2] + -12.908;
   1:  PR[91,3] = PR[90,3] + 46.326;
   1:L PR[91] R[100]mm/sec CNT100;
   1:  PR[91,1] = PR[90,1] + -22.193;
   1:  PR[91,2] = PR[90,2] + -13.681;
   1:  PR[91,3] = PR[90,3] + 46.335;
   1:L PR[91] R[100]mm/sec CNT100;
   1:  PR[91,1] = PR[90,1] + -21.428;
   1:  PR[91,2] = PR[90,2] + -14.418;
   1:  PR[91,3] = PR[90,3] + 46.344;
   1:L PR[91] R[100]mm/sec CNT100;
   1:  PR[91,1] = PR[90,1] + -20.625;
   1:  PR[91,2] = PR[90,2] + -15.116;
   1:  PR[91,3] = PR[90,3] + 46.353;
   1:L PR[91] R[100]mm/sec CNT100;
   1:  PR[91,1] = PR[90,1] + -19.786;
   1:  PR[91,2] = PR[90,2] + -15.775;
   1:  PR[91,3] = PR[90,3] + 46.362;
   1:L PR[91] R[100]mm/sec CNT100;
   1:  PR[91,1] = PR[90,1] + -18.913;
   1:  PR[91,2] = PR[90,2] + -16.393;
   1:  PR[91,3] = PR[90,3] + 46.371;
   1:L PR[91] R[100]mm/sec CNT100;
   1:  PR[91,1] = PR[90,1] + -18.007;
   1:  PR[91,2] = PR[90,2] + -16.968;
   1:  PR[91,3] = PR[90,3] + 46.380;
   1:L PR[91] R[100]mm/sec CNT100;
   1:  PR[91,1] = PR[90,1] + -17.071;
   1:  PR[91,2] = PR[90,2] + -17.500;
   1:  PR[91,3] = PR[90,3] + 46.389;
   1:L PR[91] R[100]mm/sec CNT100;
   1:  PR[91,1] = PR[90,1] + -16.108;
   1:  PR[91,2] = PR[90,2] + -17.986;
   1:  PR[91,3] = PR[90,3] + 46.398;
   1:L PR[91] R[100]mm/sec CNT100;
   1:  PR[91,1] = PR[90,1] + -15.120;
   1:  PR[91,2] = PR[90,2] + -18.424;
   1:  PR[91,3] = PR[90,3] + 46.407;
   1:L PR[91] R[100]mm/sec CNT100;
   1:  PR[91,1] = PR[90,1] + -14.110;
   1:  PR[91,2] = PR[90,2] + -18.813;
   1:  PR[91,3] = PR[90,3] + 46.416;
   1:L PR[91] R[100]mm/sec CNT100;
   1:  PR[91,1] = PR[90,1] + -13.080;
   1:  PR[91,2] = PR[90,2] + -19.152;
   1:  PR[91,3] = PR[90,3] + 46.425;
   1:L PR[91] R[100]mm/sec CNT100;
   1:  PR[91,1] = PR[90,1] + -12.032;
   1:  PR[91,2] = PR[90,2] + -19.440;
   1:  PR[91,3] = PR[90,3] + 46.434;
   1:L PR[91] R[100]mm/sec CNT100;
   1:  PR[91,1] = PR[90,1] + -10.970;
   1:  PR[91,2] = PR[90,2] + -19.675;
   1:  PR[91,3] = PR[90,3] + 46.443;
   1:L PR[91] R[100]mm/sec CNT100;
   1:  PR[91,1] = PR[90,1] + -9.897;
   1:  PR[91,2] = PR[90,2] + -19.857;
   1:  PR[91,3] = PR[90,3] + 46.452;
   1:L PR[91] R[100]mm/sec CNT100;
   1:  PR[91,1] = PR[90,1] + -8.814;
   1:  PR[91,2] = PR[90,2] + -19.986;
   1:  PR[91,3] = PR[90,3] + 46.462;
   1:L PR[91] R[100]mm/sec CNT100;
   1:  PR[91,1] = PR[90,1] + -7.726;
   1:  PR[91,2] = PR[90,2] + -20.060;
   1:  PR[91,3] = PR[90,3] + 46.471;
   1:L PR[91] R[100]mm/sec CNT100;
   1:  PR[91,1] = PR[90,1] + -6.635;
   1:  PR[91,2] = PR[90,2] + -20.080;
   1:  PR[91,3] = PR[90,3] + 46.480;
   1:L PR[91] R[100]mm/sec CNT100;
   1:  PR[91,1] = PR[90,1] + -5.543;
   1:  PR[91,2] = PR[90,2] + -20.045;
   1:  PR[91,3] = PR[90,3] + 46.489;
   1:L PR[91] R[100]mm/sec CNT100;
   1:  PR[91,1] = PR[90,1] + -4.455;
   1:  PR[91,2] = PR[90,2] + -19.956;
   1:  PR[91,3] = PR[90,3] + 46.498;
   1:L PR[91] R[100]mm/sec CNT100;
   1:  PR[91,1] = PR[90,1] + -3.372;
   1:  PR[91,2] = PR[90,2] + -19.812;
   1:  PR[91,3] = PR[90,3] + 46.507;
   1:L PR[91] R[100]mm/sec CNT100;
   1:  PR[91,1] = PR[90,1] + -2.297;
   1:  PR[91,2] = PR[90,2] + -19.613;
   1:  PR[91,3] = PR[90,3] + 46.517;
   1:L PR[91] R[100]mm/sec CNT100;
   1:  PR[91,1] = PR[90,1] + -1.230;
   1:  PR[91,2] = PR[90,2] + -19.359;
   1:  PR[91,3] = PR[90,3] + 46.526;
   1:L PR[91] R[100]mm/sec CNT100;
   1:  PR[91,1] = PR[90,1] + -0.909;
   1:  PR[91,2] = PR[90,2] + -19.267;
   1:  PR[91,3] = PR[90,3] + 46.535;
   1:L PR[91] R[100]mm/sec CNT100;
   1:  PR[91,1] = PR[90,1] + -0.451;
   1:  PR[91,2] = PR[90,2] + -19.178;
   1:  PR[91,3] = PR[90,3] + 46.538;
   1:L PR[91] R[100]mm/sec CNT100;
   1:  PR[91,1] = PR[90,1] + 0.039;
   1:  PR[91,2] = PR[90,2] + -19.163;
   1:  PR[91,3] = PR[90,3] + 46.542;
   1:L PR[91] R[100]mm/sec CNT100;
   1:  PR[91,1] = PR[90,1] + 0.522;
   1:  PR[91,2] = PR[90,2] + -19.230;
   1:  PR[91,3] = PR[90,3] + 46.546;
   1:L PR[91] R[100]mm/sec CNT100;
   1:  PR[91] = PR[90];
   1:  PR[91,1] = PR[90,1] + 1.535;
   1:  PR[91,2] = PR[90,2] + -19.848;
   1:  PR[91,3] = PR[90,3] + 47.880;
   1:L PR[91] R[100]mm/sec CNT100;
   1:  PR[91,1] = PR[90,1] + 2.620;
   1:  PR[91,2] = PR[90,2] + -20.048;
   1:  PR[91,3] = PR[90,3] + 46.558;
   1:L PR[91] R[100]mm/sec CNT100;
   1:  PR[91,1] = PR[90,1] + 3.714;
   1:  PR[91,2] = PR[90,2] + -20.192;
   1:  PR[91,3] = PR[90,3] + 46.568;
   1:L PR[91] R[100]mm/sec CNT100;
   1:  PR[91,1] = PR[90,1] + 4.818;
   1:  PR[91,2] = PR[90,2] + -20.280;
   1:  PR[91,3] = PR[90,3] + 46.577;
   1:L PR[91] R[100]mm/sec CNT100;
   1:  PR[91,1] = PR[90,1] + 5.914;
   1:  PR[91,2] = PR[90,2] + -20.314;
   1:  PR[91,3] = PR[90,3] + 46.586;
   1:L PR[91] R[100]mm/sec CNT100;
   1:  PR[91,1] = PR[90,1] + 7.014;
   1:  PR[91,2] = PR[90,2] + -20.294;
   1:  PR[91,3] = PR[90,3] + 46.596;
   1:L PR[91] R[100]mm/sec CNT100;
   1:  PR[91,1] = PR[90,1] + 8.111;
   1:  PR[91,2] = PR[90,2] + -20.218;
   1:  PR[91,3] = PR[90,3] + 46.605;
   1:L PR[91] R[100]mm/sec CNT100;
   1:  PR[91,1] = PR[90,1] + 9.202;
   1:  PR[91,2] = PR[90,2] + -20.087;
   1:  PR[91,3] = PR[90,3] + 46.614;
   1:L PR[91] R[100]mm/sec CNT100;
   1:  PR[91,1] = PR[90,1] + 10.284;
   1:  PR[91,2] = PR[90,2] + -19.902;
   1:  PR[91,3] = PR[90,3] + 46.624;
   1:L PR[91] R[100]mm/sec CNT100;
   1:  PR[91,1] = PR[90,1] + 11.354;
   1:  PR[91,2] = PR[90,2] + -19.664;
   1:  PR[91,3] = PR[90,3] + 46.633;
   1:L PR[91] R[100]mm/sec CNT100;
   1:  PR[91,1] = PR[90,1] + 12.409;
   1:  PR[91,2] = PR[90,2] + -19.373;
   1:  PR[91,3] = PR[90,3] + 46.642;
   1:L PR[91] R[100]mm/sec CNT100;
   1:  PR[91,1] = PR[90,1] + 13.448;
   1:  PR[91,2] = PR[90,2] + -19.030;
   1:  PR[91,3] = PR[90,3] + 46.651;
   1:L PR[91] R[100]mm/sec CNT100;
   1:  PR[91,1] = PR[90,1] + 14.467;
   1:  PR[91,2] = PR[90,2] + -18.636;
   1:  PR[91,3] = PR[90,3] + 46.661;
   1:L PR[91] R[100]mm/sec CNT100;
   1:  PR[91,1] = PR[90,1] + 15.462;
   1:  PR[91,2] = PR[90,2] + -18.194;
   1:  PR[91,3] = PR[90,3] + 46.670;
   1:L PR[91] R[100]mm/sec CNT100;
   1:  PR[91,1] = PR[90,1] + 16.433;
   1:  PR[91,2] = PR[90,2] + -17.703;
   1:  PR[91,3] = PR[90,3] + 46.679;
   1:L PR[91] R[100]mm/sec CNT100;
   1:  PR[91,1] = PR[90,1] + 17.376;
   1:  PR[91,2] = PR[90,2] + -17.166;
   1:  PR[91,3] = PR[90,3] + 46.688;
   1:L PR[91] R[100]mm/sec CNT100;
   1:  PR[91,1] = PR[90,1] + 18.289;
   1:  PR[91,2] = PR[90,2] + -16.583;
   1:  PR[91,3] = PR[90,3] + 46.697;
   1:L PR[91] R[100]mm/sec CNT100;
   1:  PR[91,1] = PR[90,1] + 19.169;
   1:  PR[91,2] = PR[90,2] + -15.957;
   1:  PR[91,3] = PR[90,3] + 46.707;
   1:L PR[91] R[100]mm/sec CNT100;
   1:  PR[91,1] = PR[90,1] + 20.015;
   1:  PR[91,2] = PR[90,2] + -15.289;
   1:  PR[91,3] = PR[90,3] + 46.716;
   1:L PR[91] R[100]mm/sec CNT100;
   1:  PR[91,1] = PR[90,1] + 20.824;
   1:  PR[91,2] = PR[90,2] + -14.581;
   1:  PR[91,3] = PR[90,3] + 46.725;
   1:L PR[91] R[100]mm/sec CNT100;
   1:  PR[91,1] = PR[90,1] + 21.594;
   1:  PR[91,2] = PR[90,2] + -13.834;
   1:  PR[91,3] = PR[90,3] + 46.734;
   1:L PR[91] R[100]mm/sec CNT100;
   1:  PR[91,1] = PR[90,1] + 22.324;
   1:  PR[91,2] = PR[90,2] + -13.050;
   1:  PR[91,3] = PR[90,3] + 46.743;
   1:L PR[91] R[100]mm/sec CNT100;
   1:  PR[91,1] = PR[90,1] + 23.011;
   1:  PR[91,2] = PR[90,2] + -12.231;
   1:  PR[91,3] = PR[90,3] + 46.752;
   1:L PR[91] R[100]mm/sec CNT100;
   1:  PR[91,1] = PR[90,1] + 23.654;
   1:  PR[91,2] = PR[90,2] + -11.380;
   1:  PR[91,3] = PR[90,3] + 46.761;
   1:L PR[91] R[100]mm/sec CNT100;
   1:  PR[91,1] = PR[90,1] + 24.252;
   1:  PR[91,2] = PR[90,2] + -10.498;
   1:  PR[91,3] = PR[90,3] + 46.770;
   1:L PR[91] R[100]mm/sec CNT100;
   1:  PR[91,1] = PR[90,1] + 24.802;
   1:  PR[91,2] = PR[90,2] + -9.590;
   1:  PR[91,3] = PR[90,3] + 46.779;
   1:L PR[91] R[100]mm/sec CNT100;
   1:  PR[91,1] = PR[90,1] + 25.305;
   1:  PR[91,2] = PR[90,2] + -8.658;
   1:  PR[91,3] = PR[90,3] + 46.788;
   1:L PR[91] R[100]mm/sec CNT100;
   1:  PR[91,1] = PR[90,1] + 25.757;
   1:  PR[91,2] = PR[90,2] + -7.706;
   1:  PR[91,3] = PR[90,3] + 46.797;
   1:L PR[91] R[100]mm/sec CNT100;
   1:  PR[91,1] = PR[90,1] + 26.159;
   1:  PR[91,2] = PR[90,2] + -6.739;
   1:  PR[91,3] = PR[90,3] + 46.806;
   1:L PR[91] R[100]mm/sec CNT100;
   1:  PR[91,1] = PR[90,1] + 26.509;
   1:  PR[91,2] = PR[90,2] + -5.758;
   1:  PR[91,3] = PR[90,3] + 46.815;
   1:L PR[91] R[100]mm/sec CNT100;
   1:  PR[91,1] = PR[90,1] + 26.807;
   1:  PR[91,2] = PR[90,2] + -4.764;
   1:  PR[91,3] = PR[90,3] + 46.824;
   1:L PR[91] R[100]mm/sec CNT100;
   1:  PR[91,1] = PR[90,1] + 27.051;
   1:  PR[91,2] = PR[90,2] + -3.757;
   1:  PR[91,3] = PR[90,3] + 46.832;
   1:L PR[91] R[100]mm/sec CNT100;
   1:  PR[91,1] = PR[90,1] + 27.241;
   1:  PR[91,2] = PR[90,2] + -2.736;
   1:  PR[91,3] = PR[90,3] + 46.841;
   1:L PR[91] R[100]mm/sec CNT100;
   1:  PR[91,1] = PR[90,1] + 27.378;
   1:  PR[91,2] = PR[90,2] + -1.699;
   1:  PR[91,3] = PR[90,3] + 46.850;
   1:L PR[91] R[100]mm/sec CNT100;
   1:  PR[91,1] = PR[90,1] + 27.460;
   1:  PR[91,2] = PR[90,2] + -0.645;
   1:  PR[91,3] = PR[90,3] + 46.859;
   1:L PR[91] R[100]mm/sec CNT100;
   1:  PR[91,1] = PR[90,1] + 27.487;
   1:  PR[91,2] = PR[90,2] + 0.428;
   1:  PR[91,3] = PR[90,3] + 46.868;
   1:L PR[91] R[100]mm/sec CNT100;
   1:  PR[91,1] = PR[90,1] + 27.460;
   1:  PR[91,2] = PR[90,2] + 1.500;
   1:  PR[91,3] = PR[90,3] + 46.877;
   1:L PR[91] R[100]mm/sec CNT100;
   1:  PR[91,1] = PR[90,1] + 27.378;
   1:  PR[91,2] = PR[90,2] + 2.554;
   1:  PR[91,3] = PR[90,3] + 46.886;
   1:L PR[91] R[100]mm/sec CNT100;
   1:  PR[91,1] = PR[90,1] + 27.241;
   1:  PR[91,2] = PR[90,2] + 3.591;
   1:  PR[91,3] = PR[90,3] + 46.895;
   1:L PR[91] R[100]mm/sec CNT100;
   1:  PR[91,1] = PR[90,1] + 27.051;
   1:  PR[91,2] = PR[90,2] + 4.612;
   1:  PR[91,3] = PR[90,3] + 46.904;
   1:L PR[91] R[100]mm/sec CNT100;
   1:  PR[91,1] = PR[90,1] + 26.807;
   1:  PR[91,2] = PR[90,2] + 5.619;
   1:  PR[91,3] = PR[90,3] + 46.912;
   1:L PR[91] R[100]mm/sec CNT100;
   1:  PR[91,1] = PR[90,1] + 26.509;
   1:  PR[91,2] = PR[90,2] + 6.613;
   1:  PR[91,3] = PR[90,3] + 46.921;
   1:L PR[91] R[100]mm/sec CNT100;
   1:  PR[91,1] = PR[90,1] + 26.159;
   1:  PR[91,2] = PR[90,2] + 7.594;
   1:  PR[91,3] = PR[90,3] + 46.930;
   1:L PR[91] R[100]mm/sec CNT100;
   1:  PR[91,1] = PR[90,1] + 25.757;
   1:  PR[91,2] = PR[90,2] + 8.561;
   1:  PR[91,3] = PR[90,3] + 46.939;
   1:L PR[91] R[100]mm/sec CNT100;
   1:  PR[91,1] = PR[90,1] + 25.305;
   1:  PR[91,2] = PR[90,2] + 9.512;
   1:  PR[91,3] = PR[90,3] + 46.947;
   1:L PR[91] R[100]mm/sec CNT100;
   1:  PR[91,1] = PR[90,1] + 24.802;
   1:  PR[91,2] = PR[90,2] + 10.444;
   1:  PR[91,3] = PR[90,3] + 46.956;
   1:L PR[91] R[100]mm/sec CNT100;
   1:  PR[91,1] = PR[90,1] + 24.252;
   1:  PR[91,2] = PR[90,2] + 11.353;
   1:  PR[91,3] = PR[90,3] + 46.965;
   1:L PR[91] R[100]mm/sec CNT100;
   1:  PR[91,1] = PR[90,1] + 23.654;
   1:  PR[91,2] = PR[90,2] + 12.234;
   1:  PR[91,3] = PR[90,3] + 46.974;
   1:L PR[91] R[100]mm/sec CNT100;
   1:  PR[91,1] = PR[90,1] + 23.011;
   1:  PR[91,2] = PR[90,2] + 13.086;
   1:  PR[91,3] = PR[90,3] + 46.983;
   1:L PR[91] R[100]mm/sec CNT100;
   1:  PR[91,1] = PR[90,1] + 22.324;
   1:  PR[91,2] = PR[90,2] + 13.905;
   1:  PR[91,3] = PR[90,3] + 46.992;
   1:L PR[91] R[100]mm/sec CNT100;
   1:  PR[91,1] = PR[90,1] + 21.595;
   1:  PR[91,2] = PR[90,2] + 14.689;
   1:  PR[91,3] = PR[90,3] + 47.001;
   1:L PR[91] R[100]mm/sec CNT100;
   1:  PR[91,1] = PR[90,1] + 20.824;
   1:  PR[91,2] = PR[90,2] + 15.436;
   1:  PR[91,3] = PR[90,3] + 47.010;
   1:L PR[91] R[100]mm/sec CNT100;
   1:  PR[91,1] = PR[90,1] + 20.016;
   1:  PR[91,2] = PR[90,2] + 16.144;
   1:  PR[91,3] = PR[90,3] + 47.019;
   1:L PR[91] R[100]mm/sec CNT100;
   1:  PR[91,1] = PR[90,1] + 19.170;
   1:  PR[91,2] = PR[90,2] + 16.812;
   1:  PR[91,3] = PR[90,3] + 47.029;
   1:L PR[91] R[100]mm/sec CNT100;
   1:  PR[91,1] = PR[90,1] + 18.290;
   1:  PR[91,2] = PR[90,2] + 17.438;
   1:  PR[91,3] = PR[90,3] + 47.038;
   1:L PR[91] R[100]mm/sec CNT100;
   1:  PR[91,1] = PR[90,1] + 17.377;
   1:  PR[91,2] = PR[90,2] + 18.020;
   1:  PR[91,3] = PR[90,3] + 47.047;
   1:L PR[91] R[100]mm/sec CNT100;
   1:  PR[91,1] = PR[90,1] + 16.434;
   1:  PR[91,2] = PR[90,2] + 18.558;
   1:  PR[91,3] = PR[90,3] + 47.056;
   1:L PR[91] R[100]mm/sec CNT100;
   1:  PR[91,1] = PR[90,1] + 15.464;
   1:  PR[91,2] = PR[90,2] + 19.048;
   1:  PR[91,3] = PR[90,3] + 47.065;
   1:L PR[91] R[100]mm/sec CNT100;
   1:  PR[91,1] = PR[90,1] + 14.467;
   1:  PR[91,2] = PR[90,2] + 19.491;
   1:  PR[91,3] = PR[90,3] + 47.074;
   1:L PR[91] R[100]mm/sec CNT100;
   1:  PR[91,1] = PR[90,1] + 13.449;
   1:  PR[91,2] = PR[90,2] + 19.885;
   1:  PR[91,3] = PR[90,3] + 47.083;
   1:L PR[91] R[100]mm/sec CNT100;
   1:  PR[91,1] = PR[90,1] + 12.411;
   1:  PR[91,2] = PR[90,2] + 20.227;
   1:  PR[91,3] = PR[90,3] + 47.093;
   1:L PR[91] R[100]mm/sec CNT100;
   1:  PR[91,1] = PR[90,1] + 11.355;
   1:  PR[91,2] = PR[90,2] + 20.519;
   1:  PR[91,3] = PR[90,3] + 47.102;
   1:L PR[91] R[100]mm/sec CNT100;
   1:  PR[91,1] = PR[90,1] + 10.285;
   1:  PR[91,2] = PR[90,2] + 20.757;
   1:  PR[91,3] = PR[90,3] + 47.111;
   1:L PR[91] R[100]mm/sec CNT100;
   1:  PR[91,1] = PR[90,1] + 9.203;
   1:  PR[91,2] = PR[90,2] + 20.942;
   1:  PR[91,3] = PR[90,3] + 47.120;
   1:L PR[91] R[100]mm/sec CNT100;
   1:  PR[91,1] = PR[90,1] + 8.113;
   1:  PR[91,2] = PR[90,2] + 21.073;
   1:  PR[91,3] = PR[90,3] + 47.130;
   1:L PR[91] R[100]mm/sec CNT100;
   1:  PR[91,1] = PR[90,1] + 7.016;
   1:  PR[91,2] = PR[90,2] + 21.149;
   1:  PR[91,3] = PR[90,3] + 47.139;
   1:L PR[91] R[100]mm/sec CNT100;
   1:  PR[91,1] = PR[90,1] + 5.916;
   1:  PR[91,2] = PR[90,2] + 21.170;
   1:  PR[91,3] = PR[90,3] + 47.148;
   1:L PR[91] R[100]mm/sec CNT100;
   1:  PR[91,1] = PR[90,1] + 4.816;
   1:  PR[91,2] = PR[90,2] + 21.135;
   1:  PR[91,3] = PR[90,3] + 47.158;
   1:L PR[91] R[100]mm/sec CNT100;
   1:  PR[91,1] = PR[90,1] + 3.716;
   1:  PR[91,2] = PR[90,2] + 21.047;
   1:  PR[91,3] = PR[90,3] + 47.167;
   1:L PR[91] R[100]mm/sec CNT100;
   1:  PR[91,1] = PR[90,1] + 2.623;
   1:  PR[91,2] = PR[90,2] + 20.903;
   1:  PR[91,3] = PR[90,3] + 47.176;
   1:L PR[91] R[100]mm/sec CNT100;
   1:  PR[91,1] = PR[90,1] + 1.537;
   1:  PR[91,2] = PR[90,2] + 20.704;
   1:  PR[91,3] = PR[90,3] + 47.186;
   1:L PR[91] R[100]mm/sec CNT100;
   1:  PR[91,1] = PR[90,1] + 0.566;
   1:  PR[91,2] = PR[90,2] + 20.475;
   1:  PR[91,3] = PR[90,3] + 47.195;
   1:L PR[91] R[100]mm/sec CNT100;
   1:  PR[91,1] = PR[90,1] + 0.107;
   1:  PR[91,2] = PR[90,2] + 20.403;
   1:  PR[91,3] = PR[90,3] + 47.203;
   1:L PR[91] R[100]mm/sec CNT100;
   1:  PR[91,1] = PR[90,1] + -0.382;
   1:  PR[91,2] = PR[90,2] + 20.406;
   1:  PR[91,3] = PR[90,3] + 47.207;
   1:L PR[91] R[100]mm/sec CNT100;
   1:  PR[91,1] = PR[90,1] + -0.834;
   1:  PR[91,2] = PR[90,2] + 20.483;
   1:  PR[91,3] = PR[90,3] + 47.211;
   1:L PR[91] R[100]mm/sec CNT100;
   1:  PR[91,1] = PR[90,1] + -1.772;
   1:  PR[91,2] = PR[90,2] + 20.704;
   1:  PR[91,3] = PR[90,3] + 47.215;
   1:L PR[91] R[100]mm/sec CNT100;
   1:  PR[91,1] = PR[90,1] + -2.858;
   1:  PR[91,2] = PR[90,2] + 20.903;
   1:  PR[91,3] = PR[90,3] + 47.223;
   1:L PR[91] R[100]mm/sec CNT100;
   1:  PR[91,1] = PR[90,1] + -3.952;
   1:  PR[91,2] = PR[90,2] + 21.047;
   1:  PR[91,3] = PR[90,3] + 47.233;
   1:L PR[91] R[100]mm/sec CNT100;
   1:  PR[91,1] = PR[90,1] + -5.056;
   1:  PR[91,2] = PR[90,2] + 21.135;
   1:  PR[91,3] = PR[90,3] + 47.242;
   1:L PR[91] R[100]mm/sec CNT100;
   1:  PR[91,1] = PR[90,1] + -6.152;
   1:  PR[91,2] = PR[90,2] + 21.169;
   1:  PR[91,3] = PR[90,3] + 47.251;
   1:L PR[91] R[100]mm/sec CNT100;
   1:  PR[91,1] = PR[90,1] + -7.252;
   1:  PR[91,2] = PR[90,2] + 21.149;
   1:  PR[91,3] = PR[90,3] + 47.261;
   1:L PR[91] R[100]mm/sec CNT100;
   1:  PR[91,1] = PR[90,1] + -8.349;
   1:  PR[91,2] = PR[90,2] + 21.073;
   1:  PR[91,3] = PR[90,3] + 47.270;
   1:L PR[91] R[100]mm/sec CNT100;
   1:  PR[91,1] = PR[90,1] + -9.440;
   1:  PR[91,2] = PR[90,2] + 20.942;
   1:  PR[91,3] = PR[90,3] + 47.279;
   1:L PR[91] R[100]mm/sec CNT100;
   1:  PR[91,1] = PR[90,1] + -10.522;
   1:  PR[91,2] = PR[90,2] + 20.757;
   1:  PR[91,3] = PR[90,3] + 47.289;
   1:L PR[91] R[100]mm/sec CNT100;
   1:  PR[91,1] = PR[90,1] + -11.592;
   1:  PR[91,2] = PR[90,2] + 20.519;
   1:  PR[91,3] = PR[90,3] + 47.298;
   1:L PR[91] R[100]mm/sec CNT100;
   1:  PR[91,1] = PR[90,1] + -12.648;
   1:  PR[91,2] = PR[90,2] + 20.229;
   1:  PR[91,3] = PR[90,3] + 47.307;
   1:L PR[91] R[100]mm/sec CNT100;
   1:  PR[91,1] = PR[90,1] + -13.686;
   1:  PR[91,2] = PR[90,2] + 19.886;
   1:  PR[91,3] = PR[90,3] + 47.316;
   1:L PR[91] R[100]mm/sec CNT100;
   1:  PR[91,1] = PR[90,1] + -14.705;
   1:  PR[91,2] = PR[90,2] + 19.492;
   1:  PR[91,3] = PR[90,3] + 47.326;
   1:L PR[91] R[100]mm/sec CNT100;
   1:  PR[91,1] = PR[90,1] + -15.700;
   1:  PR[91,2] = PR[90,2] + 19.049;
   1:  PR[91,3] = PR[90,3] + 47.335;
   1:L PR[91] R[100]mm/sec CNT100;
   1:  PR[91,1] = PR[90,1] + -16.671;
   1:  PR[91,2] = PR[90,2] + 18.558;
   1:  PR[91,3] = PR[90,3] + 47.344;
   1:L PR[91] R[100]mm/sec CNT100;
   1:  PR[91,1] = PR[90,1] + -17.614;
   1:  PR[91,2] = PR[90,2] + 18.020;
   1:  PR[91,3] = PR[90,3] + 47.353;
   1:L PR[91] R[100]mm/sec CNT100;
   1:  PR[91,1] = PR[90,1] + -18.527;
   1:  PR[91,2] = PR[90,2] + 17.437;
   1:  PR[91,3] = PR[90,3] + 47.362;
   1:L PR[91] R[100]mm/sec CNT100;
   1:  PR[91,1] = PR[90,1] + -19.408;
   1:  PR[91,2] = PR[90,2] + 16.811;
   1:  PR[91,3] = PR[90,3] + 47.372;
   1:L PR[91] R[100]mm/sec CNT100;
   1:  PR[91,1] = PR[90,1] + -20.253;
   1:  PR[91,2] = PR[90,2] + 16.143;
   1:  PR[91,3] = PR[90,3] + 47.381;
   1:L PR[91] R[100]mm/sec CNT100;
   1:  PR[91,1] = PR[90,1] + -21.062;
   1:  PR[91,2] = PR[90,2] + 15.435;
   1:  PR[91,3] = PR[90,3] + 47.390;
   1:L PR[91] R[100]mm/sec CNT100;
   1:  PR[91,1] = PR[90,1] + -21.833;
   1:  PR[91,2] = PR[90,2] + 14.689;
   1:  PR[91,3] = PR[90,3] + 47.399;
   1:L PR[91] R[100]mm/sec CNT100;
   1:  PR[91,1] = PR[90,1] + -22.562;
   1:  PR[91,2] = PR[90,2] + 13.907;
   1:  PR[91,3] = PR[90,3] + 47.408;
   1:L PR[91] R[100]mm/sec CNT100;
   1:  PR[91,1] = PR[90,1] + -23.249;
   1:  PR[91,2] = PR[90,2] + 13.089;
   1:  PR[91,3] = PR[90,3] + 47.417;
   1:L PR[91] R[100]mm/sec CNT100;
   1:  PR[91,1] = PR[90,1] + -23.893;
   1:  PR[91,2] = PR[90,2] + 12.239;
   1:  PR[91,3] = PR[90,3] + 47.426;
   1:L PR[91] R[100]mm/sec CNT100;
   1:  PR[91,1] = PR[90,1] + -24.490;
   1:  PR[91,2] = PR[90,2] + 11.358;
   1:  PR[91,3] = PR[90,3] + 47.435;
   1:L PR[91] R[100]mm/sec CNT100;
   1:  PR[91,1] = PR[90,1] + -25.040;
   1:  PR[91,2] = PR[90,2] + 10.449;
   1:  PR[91,3] = PR[90,3] + 47.444;
   1:L PR[91] R[100]mm/sec CNT100;
   1:  PR[91,1] = PR[90,1] + -25.543;
   1:  PR[91,2] = PR[90,2] + 9.515;
   1:  PR[91,3] = PR[90,3] + 47.453;
   1:L PR[91] R[100]mm/sec CNT100;
   1:  PR[91,1] = PR[90,1] + -25.995;
   1:  PR[91,2] = PR[90,2] + 8.561;
   1:  PR[91,3] = PR[90,3] + 47.462;
   1:L PR[91] R[100]mm/sec CNT100;
   1:  PR[91,1] = PR[90,1] + -26.397;
   1:  PR[91,2] = PR[90,2] + 7.590;
   1:  PR[91,3] = PR[90,3] + 47.471;
   1:L PR[91] R[100]mm/sec CNT100;
   1:  PR[91,1] = PR[90,1] + -26.748;
   1:  PR[91,2] = PR[90,2] + 6.606;
   1:  PR[91,3] = PR[90,3] + 47.480;
   1:L PR[91] R[100]mm/sec CNT100;
   1:  PR[91,1] = PR[90,1] + -27.045;
   1:  PR[91,2] = PR[90,2] + 5.611;
   1:  PR[91,3] = PR[90,3] + 47.489;
   1:L PR[91] R[100]mm/sec CNT100;
   1:  PR[91,1] = PR[90,1] + -27.289;
   1:  PR[91,2] = PR[90,2] + 4.605;
   1:  PR[91,3] = PR[90,3] + 47.497;
   1:L PR[91] R[100]mm/sec CNT100;
   1:  PR[91,1] = PR[90,1] + -27.480;
   1:  PR[91,2] = PR[90,2] + 3.586;
   1:  PR[91,3] = PR[90,3] + 47.506;
   1:L PR[91] R[100]mm/sec CNT100;
   1:  PR[91,1] = PR[90,1] + -27.616;
   1:  PR[91,2] = PR[90,2] + 2.551;
   1:  PR[91,3] = PR[90,3] + 47.515;
   1:L PR[91] R[100]mm/sec CNT100;
   1:  PR[91,1] = PR[90,1] + -27.698;
   1:  PR[91,2] = PR[90,2] + 1.499;
   1:  PR[91,3] = PR[90,3] + 47.524;
   1:L PR[91] R[100]mm/sec CNT100;
   1:  PR[91,1] = PR[90,1] + -27.726;
   1:  PR[91,2] = PR[90,2] + 0.428;
   1:  PR[91,3] = PR[90,3] + 47.533;
   1:L PR[91] R[100]mm/sec CNT100;
   1:  PR[91,1] = PR[90,1] + -27.698;
   1:  PR[91,2] = PR[90,2] + -0.644;
   1:  PR[91,3] = PR[90,3] + 47.542;
   1:L PR[91] R[100]mm/sec CNT100;
   1:  PR[91,1] = PR[90,1] + -27.616;
   1:  PR[91,2] = PR[90,2] + -1.696;
   1:  PR[91,3] = PR[90,3] + 47.551;
   1:L PR[91] R[100]mm/sec CNT100;
   1:  PR[91,1] = PR[90,1] + -27.480;
   1:  PR[91,2] = PR[90,2] + -2.731;
   1:  PR[91,3] = PR[90,3] + 47.560;
   1:L PR[91] R[100]mm/sec CNT100;
   1:  PR[91,1] = PR[90,1] + -27.289;
   1:  PR[91,2] = PR[90,2] + -3.750;
   1:  PR[91,3] = PR[90,3] + 47.568;
   1:L PR[91] R[100]mm/sec CNT100;
   1:  PR[91,1] = PR[90,1] + -27.045;
   1:  PR[91,2] = PR[90,2] + -4.756;
   1:  PR[91,3] = PR[90,3] + 47.577;
   1:L PR[91] R[100]mm/sec CNT100;
   1:  PR[91,1] = PR[90,1] + -26.747;
   1:  PR[91,2] = PR[90,2] + -5.752;
   1:  PR[91,3] = PR[90,3] + 47.586;
   1:L PR[91] R[100]mm/sec CNT100;
   1:  PR[91,1] = PR[90,1] + -26.397;
   1:  PR[91,2] = PR[90,2] + -6.735;
   1:  PR[91,3] = PR[90,3] + 47.595;
   1:L PR[91] R[100]mm/sec CNT100;
   1:  PR[91,1] = PR[90,1] + -25.995;
   1:  PR[91,2] = PR[90,2] + -7.706;
   1:  PR[91,3] = PR[90,3] + 47.604;
   1:L PR[91] R[100]mm/sec CNT100;
   1:  PR[91,1] = PR[90,1] + -25.542;
   1:  PR[91,2] = PR[90,2] + -8.660;
   1:  PR[91,3] = PR[90,3] + 47.612;
   1:L PR[91] R[100]mm/sec CNT100;
   1:  PR[91,1] = PR[90,1] + -25.040;
   1:  PR[91,2] = PR[90,2] + -9.594;
   1:  PR[91,3] = PR[90,3] + 47.621;
   1:L PR[91] R[100]mm/sec CNT100;
   1:  PR[91,1] = PR[90,1] + -24.490;
   1:  PR[91,2] = PR[90,2] + -10.503;
   1:  PR[91,3] = PR[90,3] + 47.630;
   1:L PR[91] R[100]mm/sec CNT100;
   1:  PR[91,1] = PR[90,1] + -23.892;
   1:  PR[91,2] = PR[90,2] + -11.384;
   1:  PR[91,3] = PR[90,3] + 47.639;
   1:L PR[91] R[100]mm/sec CNT100;
   1:  PR[91,1] = PR[90,1] + -23.249;
   1:  PR[91,2] = PR[90,2] + -12.234;
   1:  PR[91,3] = PR[90,3] + 47.648;
   1:L PR[91] R[100]mm/sec CNT100;
   1:  PR[91,1] = PR[90,1] + -22.562;
   1:  PR[91,2] = PR[90,2] + -13.052;
   1:  PR[91,3] = PR[90,3] + 47.657;
   1:L PR[91] R[100]mm/sec CNT100;
   1:  PR[91,1] = PR[90,1] + -21.832;
   1:  PR[91,2] = PR[90,2] + -13.835;
   1:  PR[91,3] = PR[90,3] + 47.666;
   1:L PR[91] R[100]mm/sec CNT100;
   1:  PR[91,1] = PR[90,1] + -21.062;
   1:  PR[91,2] = PR[90,2] + -14.581;
   1:  PR[91,3] = PR[90,3] + 47.675;
   1:L PR[91] R[100]mm/sec CNT100;
   1:  PR[91,1] = PR[90,1] + -20.253;
   1:  PR[91,2] = PR[90,2] + -15.288;
   1:  PR[91,3] = PR[90,3] + 47.684;
   1:L PR[91] R[100]mm/sec CNT100;
   1:  PR[91,1] = PR[90,1] + -19.407;
   1:  PR[91,2] = PR[90,2] + -15.956;
   1:  PR[91,3] = PR[90,3] + 47.694;
   1:L PR[91] R[100]mm/sec CNT100;
   1:  PR[91,1] = PR[90,1] + -18.526;
   1:  PR[91,2] = PR[90,2] + -16.583;
   1:  PR[91,3] = PR[90,3] + 47.703;
   1:L PR[91] R[100]mm/sec CNT100;
   1:  PR[91,1] = PR[90,1] + -17.613;
   1:  PR[91,2] = PR[90,2] + -17.165;
   1:  PR[91,3] = PR[90,3] + 47.712;
   1:L PR[91] R[100]mm/sec CNT100;
   1:  PR[91,1] = PR[90,1] + -16.670;
   1:  PR[91,2] = PR[90,2] + -17.703;
   1:  PR[91,3] = PR[90,3] + 47.721;
   1:L PR[91] R[100]mm/sec CNT100;
   1:  PR[91,1] = PR[90,1] + -15.699;
   1:  PR[91,2] = PR[90,2] + -18.195;
   1:  PR[91,3] = PR[90,3] + 47.730;
   1:L PR[91] R[100]mm/sec CNT100;
   1:  PR[91,1] = PR[90,1] + -14.703;
   1:  PR[91,2] = PR[90,2] + -18.638;
   1:  PR[91,3] = PR[90,3] + 47.739;
   1:L PR[91] R[100]mm/sec CNT100;
   1:  PR[91,1] = PR[90,1] + -13.685;
   1:  PR[91,2] = PR[90,2] + -19.031;
   1:  PR[91,3] = PR[90,3] + 47.749;
   1:L PR[91] R[100]mm/sec CNT100;
   1:  PR[91,1] = PR[90,1] + -12.647;
   1:  PR[91,2] = PR[90,2] + -19.374;
   1:  PR[91,3] = PR[90,3] + 47.758;
   1:L PR[91] R[100]mm/sec CNT100;
   1:  PR[91,1] = PR[90,1] + -11.591;
   1:  PR[91,2] = PR[90,2] + -19.665;
   1:  PR[91,3] = PR[90,3] + 47.767;
   1:L PR[91] R[100]mm/sec CNT100;
   1:  PR[91,1] = PR[90,1] + -10.520;
   1:  PR[91,2] = PR[90,2] + -19.903;
   1:  PR[91,3] = PR[90,3] + 47.776;
   1:L PR[91] R[100]mm/sec CNT100;
   1:  PR[91,1] = PR[90,1] + -9.438;
   1:  PR[91,2] = PR[90,2] + -20.087;
   1:  PR[91,3] = PR[90,3] + 47.786;
   1:L PR[91] R[100]mm/sec CNT100;
   1:  PR[91,1] = PR[90,1] + -8.347;
   1:  PR[91,2] = PR[90,2] + -20.218;
   1:  PR[91,3] = PR[90,3] + 47.795;
   1:L PR[91] R[100]mm/sec CNT100;
   1:  PR[91,1] = PR[90,1] + -7.251;
   1:  PR[91,2] = PR[90,2] + -20.293;
   1:  PR[91,3] = PR[90,3] + 47.804;
   1:L PR[91] R[100]mm/sec CNT100;
   1:  PR[91,1] = PR[90,1] + -6.151;
   1:  PR[91,2] = PR[90,2] + -20.314;
   1:  PR[91,3] = PR[90,3] + 47.813;
   1:L PR[91] R[100]mm/sec CNT100;
   1:  PR[91,1] = PR[90,1] + -5.050;
   1:  PR[91,2] = PR[90,2] + -20.280;
   1:  PR[91,3] = PR[90,3] + 47.823;
   1:L PR[91] R[100]mm/sec CNT100;
   1:  PR[91,1] = PR[90,1] + -3.950;
   1:  PR[91,2] = PR[90,2] + -20.191;
   1:  PR[91,3] = PR[90,3] + 47.832;
   1:L PR[91] R[100]mm/sec CNT100;
   1:  PR[91,1] = PR[90,1] + -2.857;
   1:  PR[91,2] = PR[90,2] + -20.047;
   1:  PR[91,3] = PR[90,3] + 47.841;
   1:L PR[91] R[100]mm/sec CNT100;
   1:  PR[91,1] = PR[90,1] + -1.770;
   1:  PR[91,2] = PR[90,2] + -19.848;
   1:  PR[91,3] = PR[90,3] + 47.851;
   1:L PR[91] R[100]mm/sec CNT100;
   1:  PR[91,1] = PR[90,1] + -0.834;
   1:  PR[91,2] = PR[90,2] + -19.628;
   1:  PR[91,3] = PR[90,3] + 47.860;
   1:L PR[91] R[100]mm/sec CNT100;
   1:  PR[91,1] = PR[90,1] + -0.382;
   1:  PR[91,2] = PR[90,2] + -19.551;
   1:  PR[91,3] = PR[90,3] + 47.868;
   1:L PR[91] R[100]mm/sec CNT100;
   1:  PR[91,1] = PR[90,1] + 0.107;
   1:  PR[91,2] = PR[90,2] + -19.548;
   1:  PR[91,3] = PR[90,3] + 47.872;
   1:L PR[91] R[100]mm/sec CNT100;
   1:  PR[91,1] = PR[90,1] + 0.566;
   1:  PR[91,2] = PR[90,2] + -19.620;
   1:  PR[91,3] = PR[90,3] + 47.876;
   1:L PR[91] R[100]mm/sec CNT100;
   1:  PR[91] = PR[90];
   1:  PR[91,1] = PR[90,1] + 2.086;
   1:  PR[91,2] = PR[90,2] + -20.293;
   1:  PR[91,3] = PR[90,3] + 49.210;
   1:L PR[91] R[100]mm/sec CNT100;
   1:  PR[91,1] = PR[90,1] + 3.187;
   1:  PR[91,2] = PR[90,2] + -20.439;
   1:  PR[91,3] = PR[90,3] + 47.896;
   1:L PR[91] R[100]mm/sec CNT100;
   1:  PR[91,1] = PR[90,1] + 4.296;
   1:  PR[91,2] = PR[90,2] + -20.529;
   1:  PR[91,3] = PR[90,3] + 47.906;
   1:L PR[91] R[100]mm/sec CNT100;
   1:  PR[91,1] = PR[90,1] + 5.408;
   1:  PR[91,2] = PR[90,2] + -20.563;
   1:  PR[91,3] = PR[90,3] + 47.915;
   1:L PR[91] R[100]mm/sec CNT100;
   1:  PR[91,1] = PR[90,1] + 6.520;
   1:  PR[91,2] = PR[90,2] + -20.541;
   1:  PR[91,3] = PR[90,3] + 47.925;
   1:L PR[91] R[100]mm/sec CNT100;
   1:  PR[91,1] = PR[90,1] + 7.628;
   1:  PR[91,2] = PR[90,2] + -20.463;
   1:  PR[91,3] = PR[90,3] + 47.934;
   1:L PR[91] R[100]mm/sec CNT100;
   1:  PR[91,1] = PR[90,1] + 8.730;
   1:  PR[91,2] = PR[90,2] + -20.330;
   1:  PR[91,3] = PR[90,3] + 47.944;
   1:L PR[91] R[100]mm/sec CNT100;
   1:  PR[91,1] = PR[90,1] + 9.823;
   1:  PR[91,2] = PR[90,2] + -20.142;
   1:  PR[91,3] = PR[90,3] + 47.953;
   1:L PR[91] R[100]mm/sec CNT100;
   1:  PR[91,1] = PR[90,1] + 10.904;
   1:  PR[91,2] = PR[90,2] + -19.899;
   1:  PR[91,3] = PR[90,3] + 47.963;
   1:L PR[91] R[100]mm/sec CNT100;
   1:  PR[91,1] = PR[90,1] + 11.970;
   1:  PR[91,2] = PR[90,2] + -19.604;
   1:  PR[91,3] = PR[90,3] + 47.972;
   1:L PR[91] R[100]mm/sec CNT100;
   1:  PR[91,1] = PR[90,1] + 13.018;
   1:  PR[91,2] = PR[90,2] + -19.255;
   1:  PR[91,3] = PR[90,3] + 47.981;
   1:L PR[91] R[100]mm/sec CNT100;
   1:  PR[91,1] = PR[90,1] + 14.046;
   1:  PR[91,2] = PR[90,2] + -18.856;
   1:  PR[91,3] = PR[90,3] + 47.991;
   1:L PR[91] R[100]mm/sec CNT100;
   1:  PR[91,1] = PR[90,1] + 15.051;
   1:  PR[91,2] = PR[90,2] + -18.407;
   1:  PR[91,3] = PR[90,3] + 48.000;
   1:L PR[91] R[100]mm/sec CNT100;
   1:  PR[91,1] = PR[90,1] + 16.031;
   1:  PR[91,2] = PR[90,2] + -17.909;
   1:  PR[91,3] = PR[90,3] + 48.009;
   1:L PR[91] R[100]mm/sec CNT100;
   1:  PR[91,1] = PR[90,1] + 16.982;
   1:  PR[91,2] = PR[90,2] + -17.364;
   1:  PR[91,3] = PR[90,3] + 48.019;
   1:L PR[91] R[100]mm/sec CNT100;
   1:  PR[91,1] = PR[90,1] + 17.903;
   1:  PR[91,2] = PR[90,2] + -16.774;
   1:  PR[91,3] = PR[90,3] + 48.028;
   1:L PR[91] R[100]mm/sec CNT100;
   1:  PR[91,1] = PR[90,1] + 18.790;
   1:  PR[91,2] = PR[90,2] + -16.142;
   1:  PR[91,3] = PR[90,3] + 48.037;
   1:L PR[91] R[100]mm/sec CNT100;
   1:  PR[91,1] = PR[90,1] + 19.643;
   1:  PR[91,2] = PR[90,2] + -15.466;
   1:  PR[91,3] = PR[90,3] + 48.047;
   1:L PR[91] R[100]mm/sec CNT100;
   1:  PR[91,1] = PR[90,1] + 20.459;
   1:  PR[91,2] = PR[90,2] + -14.750;
   1:  PR[91,3] = PR[90,3] + 48.056;
   1:L PR[91] R[100]mm/sec CNT100;
   1:  PR[91,1] = PR[90,1] + 21.235;
   1:  PR[91,2] = PR[90,2] + -13.995;
   1:  PR[91,3] = PR[90,3] + 48.065;
   1:L PR[91] R[100]mm/sec CNT100;
   1:  PR[91,1] = PR[90,1] + 21.971;
   1:  PR[91,2] = PR[90,2] + -13.203;
   1:  PR[91,3] = PR[90,3] + 48.074;
   1:L PR[91] R[100]mm/sec CNT100;
   1:  PR[91,1] = PR[90,1] + 22.664;
   1:  PR[91,2] = PR[90,2] + -12.375;
   1:  PR[91,3] = PR[90,3] + 48.083;
   1:L PR[91] R[100]mm/sec CNT100;
   1:  PR[91,1] = PR[90,1] + 23.312;
   1:  PR[91,2] = PR[90,2] + -11.515;
   1:  PR[91,3] = PR[90,3] + 48.093;
   1:L PR[91] R[100]mm/sec CNT100;
   1:  PR[91,1] = PR[90,1] + 23.915;
   1:  PR[91,2] = PR[90,2] + -10.624;
   1:  PR[91,3] = PR[90,3] + 48.102;
   1:L PR[91] R[100]mm/sec CNT100;
   1:  PR[91,1] = PR[90,1] + 24.471;
   1:  PR[91,2] = PR[90,2] + -9.705;
   1:  PR[91,3] = PR[90,3] + 48.111;
   1:L PR[91] R[100]mm/sec CNT100;
   1:  PR[91,1] = PR[90,1] + 24.977;
   1:  PR[91,2] = PR[90,2] + -8.763;
   1:  PR[91,3] = PR[90,3] + 48.120;
   1:L PR[91] R[100]mm/sec CNT100;
   1:  PR[91,1] = PR[90,1] + 25.434;
   1:  PR[91,2] = PR[90,2] + -7.801;
   1:  PR[91,3] = PR[90,3] + 48.129;
   1:L PR[91] R[100]mm/sec CNT100;
   1:  PR[91,1] = PR[90,1] + 25.839;
   1:  PR[91,2] = PR[90,2] + -6.822;
   1:  PR[91,3] = PR[90,3] + 48.138;
   1:L PR[91] R[100]mm/sec CNT100;
   1:  PR[91,1] = PR[90,1] + 26.192;
   1:  PR[91,2] = PR[90,2] + -5.829;
   1:  PR[91,3] = PR[90,3] + 48.147;
   1:L PR[91] R[100]mm/sec CNT100;
   1:  PR[91,1] = PR[90,1] + 26.492;
   1:  PR[91,2] = PR[90,2] + -4.822;
   1:  PR[91,3] = PR[90,3] + 48.156;
   1:L PR[91] R[100]mm/sec CNT100;
   1:  PR[91,1] = PR[90,1] + 26.739;
   1:  PR[91,2] = PR[90,2] + -3.802;
   1:  PR[91,3] = PR[90,3] + 48.165;
   1:L PR[91] R[100]mm/sec CNT100;
   1:  PR[91,1] = PR[90,1] + 26.931;
   1:  PR[91,2] = PR[90,2] + -2.768;
   1:  PR[91,3] = PR[90,3] + 48.174;
   1:L PR[91] R[100]mm/sec CNT100;
   1:  PR[91,1] = PR[90,1] + 27.069;
   1:  PR[91,2] = PR[90,2] + -1.718;
   1:  PR[91,3] = PR[90,3] + 48.183;
   1:L PR[91] R[100]mm/sec CNT100;
   1:  PR[91,1] = PR[90,1] + 27.151;
   1:  PR[91,2] = PR[90,2] + -0.655;
   1:  PR[91,3] = PR[90,3] + 48.192;
   1:L PR[91] R[100]mm/sec CNT100;
   1:  PR[91,1] = PR[90,1] + 27.176;
   1:  PR[91,2] = PR[90,2] + 0.428;
   1:  PR[91,3] = PR[90,3] + 48.201;
   1:L PR[91] R[100]mm/sec CNT100;
   1:  PR[91,1] = PR[90,1] + 27.151;
   1:  PR[91,2] = PR[90,2] + 1.510;
   1:  PR[91,3] = PR[90,3] + 48.210;
   1:L PR[91] R[100]mm/sec CNT100;
   1:  PR[91,1] = PR[90,1] + 27.069;
   1:  PR[91,2] = PR[90,2] + 2.573;
   1:  PR[91,3] = PR[90,3] + 48.219;
   1:L PR[91] R[100]mm/sec CNT100;
   1:  PR[91,1] = PR[90,1] + 26.931;
   1:  PR[91,2] = PR[90,2] + 3.622;
   1:  PR[91,3] = PR[90,3] + 48.228;
   1:L PR[91] R[100]mm/sec CNT100;
   1:  PR[91,1] = PR[90,1] + 26.739;
   1:  PR[91,2] = PR[90,2] + 4.657;
   1:  PR[91,3] = PR[90,3] + 48.237;
   1:L PR[91] R[100]mm/sec CNT100;
   1:  PR[91,1] = PR[90,1] + 26.493;
   1:  PR[91,2] = PR[90,2] + 5.676;
   1:  PR[91,3] = PR[90,3] + 48.246;
   1:L PR[91] R[100]mm/sec CNT100;
   1:  PR[91,1] = PR[90,1] + 26.192;
   1:  PR[91,2] = PR[90,2] + 6.683;
   1:  PR[91,3] = PR[90,3] + 48.255;
   1:L PR[91] R[100]mm/sec CNT100;
   1:  PR[91,1] = PR[90,1] + 25.839;
   1:  PR[91,2] = PR[90,2] + 7.677;
   1:  PR[91,3] = PR[90,3] + 48.264;
   1:L PR[91] R[100]mm/sec CNT100;
   1:  PR[91,1] = PR[90,1] + 25.434;
   1:  PR[91,2] = PR[90,2] + 8.656;
   1:  PR[91,3] = PR[90,3] + 48.273;
   1:L PR[91] R[100]mm/sec CNT100;
   1:  PR[91,1] = PR[90,1] + 24.977;
   1:  PR[91,2] = PR[90,2] + 9.618;
   1:  PR[91,3] = PR[90,3] + 48.282;
   1:L PR[91] R[100]mm/sec CNT100;
   1:  PR[91,1] = PR[90,1] + 24.471;
   1:  PR[91,2] = PR[90,2] + 10.560;
   1:  PR[91,3] = PR[90,3] + 48.291;
   1:L PR[91] R[100]mm/sec CNT100;
   1:  PR[91,1] = PR[90,1] + 23.916;
   1:  PR[91,2] = PR[90,2] + 11.478;
   1:  PR[91,3] = PR[90,3] + 48.300;
   1:L PR[91] R[100]mm/sec CNT100;
   1:  PR[91,1] = PR[90,1] + 23.313;
   1:  PR[91,2] = PR[90,2] + 12.369;
   1:  PR[91,3] = PR[90,3] + 48.309;
   1:L PR[91] R[100]mm/sec CNT100;
   1:  PR[91,1] = PR[90,1] + 22.664;
   1:  PR[91,2] = PR[90,2] + 13.230;
   1:  PR[91,3] = PR[90,3] + 48.318;
   1:L PR[91] R[100]mm/sec CNT100;
   1:  PR[91,1] = PR[90,1] + 21.971;
   1:  PR[91,2] = PR[90,2] + 14.057;
   1:  PR[91,3] = PR[90,3] + 48.327;
   1:L PR[91] R[100]mm/sec CNT100;
   1:  PR[91,1] = PR[90,1] + 21.236;
   1:  PR[91,2] = PR[90,2] + 14.850;
   1:  PR[91,3] = PR[90,3] + 48.337;
   1:L PR[91] R[100]mm/sec CNT100;
   1:  PR[91,1] = PR[90,1] + 20.459;
   1:  PR[91,2] = PR[90,2] + 15.605;
   1:  PR[91,3] = PR[90,3] + 48.346;
   1:L PR[91] R[100]mm/sec CNT100;
   1:  PR[91,1] = PR[90,1] + 19.643;
   1:  PR[91,2] = PR[90,2] + 16.321;
   1:  PR[91,3] = PR[90,3] + 48.355;
   1:L PR[91] R[100]mm/sec CNT100;
   1:  PR[91,1] = PR[90,1] + 18.791;
   1:  PR[91,2] = PR[90,2] + 16.996;
   1:  PR[91,3] = PR[90,3] + 48.364;
   1:L PR[91] R[100]mm/sec CNT100;
   1:  PR[91,1] = PR[90,1] + 17.903;
   1:  PR[91,2] = PR[90,2] + 17.629;
   1:  PR[91,3] = PR[90,3] + 48.373;
   1:L PR[91] R[100]mm/sec CNT100;
   1:  PR[91,1] = PR[90,1] + 16.974;
   1:  PR[91,2] = PR[90,2] + 18.223;
   1:  PR[91,3] = PR[90,3] + 48.383;
   1:L PR[91] R[100]mm/sec CNT100;
   1:  PR[91,1] = PR[90,1] + 16.032;
   1:  PR[91,2] = PR[90,2] + 18.763;
   1:  PR[91,3] = PR[90,3] + 48.392;
   1:L PR[91] R[100]mm/sec CNT100;
   1:  PR[91,1] = PR[90,1] + 15.052;
   1:  PR[91,2] = PR[90,2] + 19.261;
   1:  PR[91,3] = PR[90,3] + 48.401;
   1:L PR[91] R[100]mm/sec CNT100;
   1:  PR[91,1] = PR[90,1] + 14.048;
   1:  PR[91,2] = PR[90,2] + 19.711;
   1:  PR[91,3] = PR[90,3] + 48.411;
   1:L PR[91] R[100]mm/sec CNT100;
   1:  PR[91,1] = PR[90,1] + 13.019;
   1:  PR[91,2] = PR[90,2] + 20.110;
   1:  PR[91,3] = PR[90,3] + 48.420;
   1:L PR[91] R[100]mm/sec CNT100;
   1:  PR[91,1] = PR[90,1] + 11.971;
   1:  PR[91,2] = PR[90,2] + 20.458;
   1:  PR[91,3] = PR[90,3] + 48.429;
   1:L PR[91] R[100]mm/sec CNT100;
   1:  PR[91,1] = PR[90,1] + 10.905;
   1:  PR[91,2] = PR[90,2] + 20.754;
   1:  PR[91,3] = PR[90,3] + 48.439;
   1:L PR[91] R[100]mm/sec CNT100;
   1:  PR[91,1] = PR[90,1] + 9.824;
   1:  PR[91,2] = PR[90,2] + 20.997;
   1:  PR[91,3] = PR[90,3] + 48.448;
   1:L PR[91] R[100]mm/sec CNT100;
   1:  PR[91,1] = PR[90,1] + 8.732;
   1:  PR[91,2] = PR[90,2] + 21.185;
   1:  PR[91,3] = PR[90,3] + 48.457;
   1:L PR[91] R[100]mm/sec CNT100;
   1:  PR[91,1] = PR[90,1] + 7.630;
   1:  PR[91,2] = PR[90,2] + 21.318;
   1:  PR[91,3] = PR[90,3] + 48.467;
   1:L PR[91] R[100]mm/sec CNT100;
   1:  PR[91,1] = PR[90,1] + 6.522;
   1:  PR[91,2] = PR[90,2] + 21.396;
   1:  PR[91,3] = PR[90,3] + 48.476;
   1:L PR[91] R[100]mm/sec CNT100;
   1:  PR[91,1] = PR[90,1] + 5.410;
   1:  PR[91,2] = PR[90,2] + 21.418;
   1:  PR[91,3] = PR[90,3] + 48.486;
   1:L PR[91] R[100]mm/sec CNT100;
   1:  PR[91,1] = PR[90,1] + 4.298;
   1:  PR[91,2] = PR[90,2] + 21.384;
   1:  PR[91,3] = PR[90,3] + 48.495;
   1:L PR[91] R[100]mm/sec CNT100;
   1:  PR[91,1] = PR[90,1] + 3.189;
   1:  PR[91,2] = PR[90,2] + 21.294;
   1:  PR[91,3] = PR[90,3] + 48.505;
   1:L PR[91] R[100]mm/sec CNT100;
   1:  PR[91,1] = PR[90,1] + 2.088;
   1:  PR[91,2] = PR[90,2] + 21.149;
   1:  PR[91,3] = PR[90,3] + 48.514;
   1:L PR[91] R[100]mm/sec CNT100;
   1:  PR[91,1] = PR[90,1] + 0.178;
   1:  PR[91,2] = PR[90,2] + 20.782;
   1:  PR[91,3] = PR[90,3] + 48.523;
   1:L PR[91] R[100]mm/sec CNT100;
   1:  PR[91,1] = PR[90,1] + -0.315;
   1:  PR[91,2] = PR[90,2] + 20.774;
   1:  PR[91,3] = PR[90,3] + 48.540;
   1:L PR[91] R[100]mm/sec CNT100;
   1:  PR[91,1] = PR[90,1] + -0.775;
   1:  PR[91,2] = PR[90,2] + 20.842;
   1:  PR[91,3] = PR[90,3] + 48.544;
   1:L PR[91] R[100]mm/sec CNT100;
   1:  PR[91,1] = PR[90,1] + -1.224;
   1:  PR[91,2] = PR[90,2] + 20.946;
   1:  PR[91,3] = PR[90,3] + 48.548;
   1:L PR[91] R[100]mm/sec CNT100;
   1:  PR[91,1] = PR[90,1] + -2.322;
   1:  PR[91,2] = PR[90,2] + 21.148;
   1:  PR[91,3] = PR[90,3] + 48.552;
   1:L PR[91] R[100]mm/sec CNT100;
   1:  PR[91,1] = PR[90,1] + -3.426;
   1:  PR[91,2] = PR[90,2] + 21.294;
   1:  PR[91,3] = PR[90,3] + 48.561;
   1:L PR[91] R[100]mm/sec CNT100;
   1:  PR[91,1] = PR[90,1] + -4.535;
   1:  PR[91,2] = PR[90,2] + 21.384;
   1:  PR[91,3] = PR[90,3] + 48.571;
   1:L PR[91] R[100]mm/sec CNT100;
   1:  PR[91,1] = PR[90,1] + -5.647;
   1:  PR[91,2] = PR[90,2] + 21.418;
   1:  PR[91,3] = PR[90,3] + 48.580;
   1:L PR[91] R[100]mm/sec CNT100;
   1:  PR[91,1] = PR[90,1] + -6.758;
   1:  PR[91,2] = PR[90,2] + 21.396;
   1:  PR[91,3] = PR[90,3] + 48.590;
   1:L PR[91] R[100]mm/sec CNT100;
   1:  PR[91,1] = PR[90,1] + -7.866;
   1:  PR[91,2] = PR[90,2] + 21.318;
   1:  PR[91,3] = PR[90,3] + 48.599;
   1:L PR[91] R[100]mm/sec CNT100;
   1:  PR[91,1] = PR[90,1] + -8.968;
   1:  PR[91,2] = PR[90,2] + 21.185;
   1:  PR[91,3] = PR[90,3] + 48.609;
   1:L PR[91] R[100]mm/sec CNT100;
   1:  PR[91,1] = PR[90,1] + -10.061;
   1:  PR[91,2] = PR[90,2] + 20.997;
   1:  PR[91,3] = PR[90,3] + 48.618;
   1:L PR[91] R[100]mm/sec CNT100;
   1:  PR[91,1] = PR[90,1] + -11.142;
   1:  PR[91,2] = PR[90,2] + 20.755;
   1:  PR[91,3] = PR[90,3] + 48.628;
   1:L PR[91] R[100]mm/sec CNT100;
   1:  PR[91,1] = PR[90,1] + -12.208;
   1:  PR[91,2] = PR[90,2] + 20.459;
   1:  PR[91,3] = PR[90,3] + 48.637;
   1:L PR[91] R[100]mm/sec CNT100;
   1:  PR[91,1] = PR[90,1] + -13.256;
   1:  PR[91,2] = PR[90,2] + 20.111;
   1:  PR[91,3] = PR[90,3] + 48.646;
   1:L PR[91] R[100]mm/sec CNT100;
   1:  PR[91,1] = PR[90,1] + -14.284;
   1:  PR[91,2] = PR[90,2] + 19.712;
   1:  PR[91,3] = PR[90,3] + 48.656;
   1:L PR[91] R[100]mm/sec CNT100;
   1:  PR[91,1] = PR[90,1] + -15.289;
   1:  PR[91,2] = PR[90,2] + 19.262;
   1:  PR[91,3] = PR[90,3] + 48.665;
   1:L PR[91] R[100]mm/sec CNT100;
   1:  PR[91,1] = PR[90,1] + -16.269;
   1:  PR[91,2] = PR[90,2] + 18.764;
   1:  PR[91,3] = PR[90,3] + 48.674;
   1:L PR[91] R[100]mm/sec CNT100;
   1:  PR[91,1] = PR[90,1] + -17.220;
   1:  PR[91,2] = PR[90,2] + 18.219;
   1:  PR[91,3] = PR[90,3] + 48.684;
   1:L PR[91] R[100]mm/sec CNT100;
   1:  PR[91,1] = PR[90,1] + -18.141;
   1:  PR[91,2] = PR[90,2] + 17.629;
   1:  PR[91,3] = PR[90,3] + 48.693;
   1:L PR[91] R[100]mm/sec CNT100;
   1:  PR[91,1] = PR[90,1] + -19.029;
   1:  PR[91,2] = PR[90,2] + 16.995;
   1:  PR[91,3] = PR[90,3] + 48.702;
   1:L PR[91] R[100]mm/sec CNT100;
   1:  PR[91,1] = PR[90,1] + -19.881;
   1:  PR[91,2] = PR[90,2] + 16.320;
   1:  PR[91,3] = PR[90,3] + 48.712;
   1:L PR[91] R[100]mm/sec CNT100;
   1:  PR[91,1] = PR[90,1] + -20.697;
   1:  PR[91,2] = PR[90,2] + 15.605;
   1:  PR[91,3] = PR[90,3] + 48.721;
   1:L PR[91] R[100]mm/sec CNT100;
   1:  PR[91,1] = PR[90,1] + -21.474;
   1:  PR[91,2] = PR[90,2] + 14.851;
   1:  PR[91,3] = PR[90,3] + 48.730;
   1:L PR[91] R[100]mm/sec CNT100;
   1:  PR[91,1] = PR[90,1] + -22.209;
   1:  PR[91,2] = PR[90,2] + 14.059;
   1:  PR[91,3] = PR[90,3] + 48.739;
   1:L PR[91] R[100]mm/sec CNT100;
   1:  PR[91,1] = PR[90,1] + -22.903;
   1:  PR[91,2] = PR[90,2] + 13.233;
   1:  PR[91,3] = PR[90,3] + 48.748;
   1:L PR[91] R[100]mm/sec CNT100;
   1:  PR[91,1] = PR[90,1] + -23.551;
   1:  PR[91,2] = PR[90,2] + 12.373;
   1:  PR[91,3] = PR[90,3] + 48.758;
   1:L PR[91] R[100]mm/sec CNT100;
   1:  PR[91,1] = PR[90,1] + -24.154;
   1:  PR[91,2] = PR[90,2] + 11.483;
   1:  PR[91,3] = PR[90,3] + 48.767;
   1:L PR[91] R[100]mm/sec CNT100;
   1:  PR[91,1] = PR[90,1] + -24.709;
   1:  PR[91,2] = PR[90,2] + 10.564;
   1:  PR[91,3] = PR[90,3] + 48.776;
   1:L PR[91] R[100]mm/sec CNT100;
   1:  PR[91,1] = PR[90,1] + -25.215;
   1:  PR[91,2] = PR[90,2] + 9.620;
   1:  PR[91,3] = PR[90,3] + 48.785;
   1:L PR[91] R[100]mm/sec CNT100;
   1:  PR[91,1] = PR[90,1] + -25.672;
   1:  PR[91,2] = PR[90,2] + 8.655;
   1:  PR[91,3] = PR[90,3] + 48.794;
   1:L PR[91] R[100]mm/sec CNT100;
   1:  PR[91,1] = PR[90,1] + -26.077;
   1:  PR[91,2] = PR[90,2] + 7.674;
   1:  PR[91,3] = PR[90,3] + 48.803;
   1:L PR[91] R[100]mm/sec CNT100;
   1:  PR[91,1] = PR[90,1] + -26.431;
   1:  PR[91,2] = PR[90,2] + 6.678;
   1:  PR[91,3] = PR[90,3] + 48.812;
   1:L PR[91] R[100]mm/sec CNT100;
   1:  PR[91,1] = PR[90,1] + -26.731;
   1:  PR[91,2] = PR[90,2] + 5.670;
   1:  PR[91,3] = PR[90,3] + 48.821;
   1:L PR[91] R[100]mm/sec CNT100;
   1:  PR[91,1] = PR[90,1] + -26.977;
   1:  PR[91,2] = PR[90,2] + 4.650;
   1:  PR[91,3] = PR[90,3] + 48.830;
   1:L PR[91] R[100]mm/sec CNT100;
   1:  PR[91,1] = PR[90,1] + -27.169;
   1:  PR[91,2] = PR[90,2] + 3.618;
   1:  PR[91,3] = PR[90,3] + 48.839;
   1:L PR[91] R[100]mm/sec CNT100;
   1:  PR[91,1] = PR[90,1] + -27.307;
   1:  PR[91,2] = PR[90,2] + 2.571;
   1:  PR[91,3] = PR[90,3] + 48.848;
   1:L PR[91] R[100]mm/sec CNT100;
   1:  PR[91,1] = PR[90,1] + -27.390;
   1:  PR[91,2] = PR[90,2] + 1.509;
   1:  PR[91,3] = PR[90,3] + 48.857;
   1:L PR[91] R[100]mm/sec CNT100;
   1:  PR[91,1] = PR[90,1] + -27.414;
   1:  PR[91,2] = PR[90,2] + 0.428;
   1:  PR[91,3] = PR[90,3] + 48.866;
   1:L PR[91] R[100]mm/sec CNT100;
   1:  PR[91,1] = PR[90,1] + -27.390;
   1:  PR[91,2] = PR[90,2] + -0.654;
   1:  PR[91,3] = PR[90,3] + 48.875;
   1:L PR[91] R[100]mm/sec CNT100;
   1:  PR[91,1] = PR[90,1] + -27.307;
   1:  PR[91,2] = PR[90,2] + -1.716;
   1:  PR[91,3] = PR[90,3] + 48.884;
   1:L PR[91] R[100]mm/sec CNT100;
   1:  PR[91,1] = PR[90,1] + -27.169;
   1:  PR[91,2] = PR[90,2] + -2.763;
   1:  PR[91,3] = PR[90,3] + 48.893;
   1:L PR[91] R[100]mm/sec CNT100;
   1:  PR[91,1] = PR[90,1] + -26.977;
   1:  PR[91,2] = PR[90,2] + -3.795;
   1:  PR[91,3] = PR[90,3] + 48.902;
   1:L PR[91] R[100]mm/sec CNT100;
   1:  PR[91,1] = PR[90,1] + -26.731;
   1:  PR[91,2] = PR[90,2] + -4.815;
   1:  PR[91,3] = PR[90,3] + 48.911;
   1:L PR[91] R[100]mm/sec CNT100;
   1:  PR[91,1] = PR[90,1] + -26.431;
   1:  PR[91,2] = PR[90,2] + -5.823;
   1:  PR[91,3] = PR[90,3] + 48.920;
   1:L PR[91] R[100]mm/sec CNT100;
   1:  PR[91,1] = PR[90,1] + -26.077;
   1:  PR[91,2] = PR[90,2] + -6.819;
   1:  PR[91,3] = PR[90,3] + 48.929;
   1:L PR[91] R[100]mm/sec CNT100;
   1:  PR[91,1] = PR[90,1] + -25.672;
   1:  PR[91,2] = PR[90,2] + -7.801;
   1:  PR[91,3] = PR[90,3] + 48.938;
   1:L PR[91] R[100]mm/sec CNT100;
   1:  PR[91,1] = PR[90,1] + -25.215;
   1:  PR[91,2] = PR[90,2] + -8.766;
   1:  PR[91,3] = PR[90,3] + 48.947;
   1:L PR[91] R[100]mm/sec CNT100;
   1:  PR[91,1] = PR[90,1] + -24.709;
   1:  PR[91,2] = PR[90,2] + -9.709;
   1:  PR[91,3] = PR[90,3] + 48.956;
   1:L PR[91] R[100]mm/sec CNT100;
   1:  PR[91,1] = PR[90,1] + -24.153;
   1:  PR[91,2] = PR[90,2] + -10.628;
   1:  PR[91,3] = PR[90,3] + 48.965;
   1:L PR[91] R[100]mm/sec CNT100;
   1:  PR[91,1] = PR[90,1] + -23.551;
   1:  PR[91,2] = PR[90,2] + -11.519;
   1:  PR[91,3] = PR[90,3] + 48.974;
   1:L PR[91] R[100]mm/sec CNT100;
   1:  PR[91,1] = PR[90,1] + -22.902;
   1:  PR[91,2] = PR[90,2] + -12.378;
   1:  PR[91,3] = PR[90,3] + 48.983;
   1:L PR[91] R[100]mm/sec CNT100;
   1:  PR[91,1] = PR[90,1] + -22.209;
   1:  PR[91,2] = PR[90,2] + -13.205;
   1:  PR[91,3] = PR[90,3] + 48.992;
   1:L PR[91] R[100]mm/sec CNT100;
   1:  PR[91,1] = PR[90,1] + -21.473;
   1:  PR[91,2] = PR[90,2] + -13.996;
   1:  PR[91,3] = PR[90,3] + 49.002;
   1:L PR[91] R[100]mm/sec CNT100;
   1:  PR[91,1] = PR[90,1] + -20.697;
   1:  PR[91,2] = PR[90,2] + -14.750;
   1:  PR[91,3] = PR[90,3] + 49.011;
   1:L PR[91] R[100]mm/sec CNT100;
   1:  PR[91,1] = PR[90,1] + -19.881;
   1:  PR[91,2] = PR[90,2] + -15.466;
   1:  PR[91,3] = PR[90,3] + 49.020;
   1:L PR[91] R[100]mm/sec CNT100;
   1:  PR[91,1] = PR[90,1] + -19.028;
   1:  PR[91,2] = PR[90,2] + -16.141;
   1:  PR[91,3] = PR[90,3] + 49.029;
   1:L PR[91] R[100]mm/sec CNT100;
   1:  PR[91,1] = PR[90,1] + -18.140;
   1:  PR[91,2] = PR[90,2] + -16.774;
   1:  PR[91,3] = PR[90,3] + 49.038;
   1:L PR[91] R[100]mm/sec CNT100;
   1:  PR[91,1] = PR[90,1] + -17.210;
   1:  PR[91,2] = PR[90,2] + -17.369;
   1:  PR[91,3] = PR[90,3] + 49.048;
   1:L PR[91] R[100]mm/sec CNT100;
   1:  PR[91,1] = PR[90,1] + -16.268;
   1:  PR[91,2] = PR[90,2] + -17.909;
   1:  PR[91,3] = PR[90,3] + 49.057;
   1:L PR[91] R[100]mm/sec CNT100;
   1:  PR[91,1] = PR[90,1] + -15.288;
   1:  PR[91,2] = PR[90,2] + -18.408;
   1:  PR[91,3] = PR[90,3] + 49.066;
   1:L PR[91] R[100]mm/sec CNT100;
   1:  PR[91,1] = PR[90,1] + -14.283;
   1:  PR[91,2] = PR[90,2] + -18.857;
   1:  PR[91,3] = PR[90,3] + 49.076;
   1:L PR[91] R[100]mm/sec CNT100;
   1:  PR[91,1] = PR[90,1] + -13.255;
   1:  PR[91,2] = PR[90,2] + -19.257;
   1:  PR[91,3] = PR[90,3] + 49.085;
   1:L PR[91] R[100]mm/sec CNT100;
   1:  PR[91,1] = PR[90,1] + -12.207;
   1:  PR[91,2] = PR[90,2] + -19.605;
   1:  PR[91,3] = PR[90,3] + 49.094;
   1:L PR[91] R[100]mm/sec CNT100;
   1:  PR[91,1] = PR[90,1] + -11.141;
   1:  PR[91,2] = PR[90,2] + -19.900;
   1:  PR[91,3] = PR[90,3] + 49.104;
   1:L PR[91] R[100]mm/sec CNT100;
   1:  PR[91,1] = PR[90,1] + -10.060;
   1:  PR[91,2] = PR[90,2] + -20.142;
   1:  PR[91,3] = PR[90,3] + 49.113;
   1:L PR[91] R[100]mm/sec CNT100;
   1:  PR[91,1] = PR[90,1] + -8.967;
   1:  PR[91,2] = PR[90,2] + -20.330;
   1:  PR[91,3] = PR[90,3] + 49.122;
   1:L PR[91] R[100]mm/sec CNT100;
   1:  PR[91,1] = PR[90,1] + -7.865;
   1:  PR[91,2] = PR[90,2] + -20.463;
   1:  PR[91,3] = PR[90,3] + 49.132;
   1:L PR[91] R[100]mm/sec CNT100;
   1:  PR[91,1] = PR[90,1] + -6.756;
   1:  PR[91,2] = PR[90,2] + -20.541;
   1:  PR[91,3] = PR[90,3] + 49.141;
   1:L PR[91] R[100]mm/sec CNT100;
   1:  PR[91,1] = PR[90,1] + -5.645;
   1:  PR[91,2] = PR[90,2] + -20.563;
   1:  PR[91,3] = PR[90,3] + 49.151;
   1:L PR[91] R[100]mm/sec CNT100;
   1:  PR[91,1] = PR[90,1] + -4.533;
   1:  PR[91,2] = PR[90,2] + -20.529;
   1:  PR[91,3] = PR[90,3] + 49.160;
   1:L PR[91] R[100]mm/sec CNT100;
   1:  PR[91,1] = PR[90,1] + -3.424;
   1:  PR[91,2] = PR[90,2] + -20.439;
   1:  PR[91,3] = PR[90,3] + 49.170;
   1:L PR[91] R[100]mm/sec CNT100;
   1:  PR[91,1] = PR[90,1] + -2.320;
   1:  PR[91,2] = PR[90,2] + -20.293;
   1:  PR[91,3] = PR[90,3] + 49.179;
   1:L PR[91] R[100]mm/sec CNT100;
   1:  PR[91,1] = PR[90,1] + -1.221;
   1:  PR[91,2] = PR[90,2] + -20.090;
   1:  PR[91,3] = PR[90,3] + 49.188;
   1:L PR[91] R[100]mm/sec CNT100;
   1:  PR[91,1] = PR[90,1] + -0.775;
   1:  PR[91,2] = PR[90,2] + -19.986;
   1:  PR[91,3] = PR[90,3] + 49.198;
   1:L PR[91] R[100]mm/sec CNT100;
   1:  PR[91,1] = PR[90,1] + -0.315;
   1:  PR[91,2] = PR[90,2] + -19.918;
   1:  PR[91,3] = PR[90,3] + 49.202;
   1:L PR[91] R[100]mm/sec CNT100;
   1:  PR[91,1] = PR[90,1] + 0.178;
   1:  PR[91,2] = PR[90,2] + -19.926;
   1:  PR[91,3] = PR[90,3] + 49.206;
   1:L PR[91] R[100]mm/sec CNT100;
   1:  PR[91] = PR[90];
   1:  PR[91,1] = PR[90,1] + 1.560;
   1:  PR[91,2] = PR[90,2] + -20.540;
   1:  PR[91,3] = PR[90,3] + 50.540;
   1:L PR[91] R[100]mm/sec CNT100;
   1:  PR[91,1] = PR[90,1] + 2.660;
   1:  PR[91,2] = PR[90,2] + -20.686;
   1:  PR[91,3] = PR[90,3] + 49.221;
   1:L PR[91] R[100]mm/sec CNT100;
   1:  PR[91,1] = PR[90,1] + 3.779;
   1:  PR[91,2] = PR[90,2] + -20.778;
   1:  PR[91,3] = PR[90,3] + 49.231;
   1:L PR[91] R[100]mm/sec CNT100;
   1:  PR[91,1] = PR[90,1] + 4.900;
   1:  PR[91,2] = PR[90,2] + -20.813;
   1:  PR[91,3] = PR[90,3] + 49.241;
   1:L PR[91] R[100]mm/sec CNT100;
   1:  PR[91,1] = PR[90,1] + 6.022;
   1:  PR[91,2] = PR[90,2] + -20.791;
   1:  PR[91,3] = PR[90,3] + 49.250;
   1:L PR[91] R[100]mm/sec CNT100;
   1:  PR[91,1] = PR[90,1] + 7.140;
   1:  PR[91,2] = PR[90,2] + -20.713;
   1:  PR[91,3] = PR[90,3] + 49.260;
   1:L PR[91] R[100]mm/sec CNT100;
   1:  PR[91,1] = PR[90,1] + 8.252;
   1:  PR[91,2] = PR[90,2] + -20.579;
   1:  PR[91,3] = PR[90,3] + 49.269;
   1:L PR[91] R[100]mm/sec CNT100;
   1:  PR[91,1] = PR[90,1] + 9.355;
   1:  PR[91,2] = PR[90,2] + -20.390;
   1:  PR[91,3] = PR[90,3] + 49.279;
   1:L PR[91] R[100]mm/sec CNT100;
   1:  PR[91,1] = PR[90,1] + 10.446;
   1:  PR[91,2] = PR[90,2] + -20.146;
   1:  PR[91,3] = PR[90,3] + 49.288;
   1:L PR[91] R[100]mm/sec CNT100;
   1:  PR[91,1] = PR[90,1] + 11.522;
   1:  PR[91,2] = PR[90,2] + -19.847;
   1:  PR[91,3] = PR[90,3] + 49.298;
   1:L PR[91] R[100]mm/sec CNT100;
   1:  PR[91,1] = PR[90,1] + 12.580;
   1:  PR[91,2] = PR[90,2] + -19.496;
   1:  PR[91,3] = PR[90,3] + 49.307;
   1:L PR[91] R[100]mm/sec CNT100;
   1:  PR[91,1] = PR[90,1] + 13.618;
   1:  PR[91,2] = PR[90,2] + -19.093;
   1:  PR[91,3] = PR[90,3] + 49.317;
   1:L PR[91] R[100]mm/sec CNT100;
   1:  PR[91,1] = PR[90,1] + 14.633;
   1:  PR[91,2] = PR[90,2] + -18.639;
   1:  PR[91,3] = PR[90,3] + 49.326;
   1:L PR[91] R[100]mm/sec CNT100;
   1:  PR[91,1] = PR[90,1] + 15.622;
   1:  PR[91,2] = PR[90,2] + -18.136;
   1:  PR[91,3] = PR[90,3] + 49.336;
   1:L PR[91] R[100]mm/sec CNT100;
   1:  PR[91,1] = PR[90,1] + 16.582;
   1:  PR[91,2] = PR[90,2] + -17.586;
   1:  PR[91,3] = PR[90,3] + 49.345;
   1:L PR[91] R[100]mm/sec CNT100;
   1:  PR[91,1] = PR[90,1] + 17.512;
   1:  PR[91,2] = PR[90,2] + -16.989;
   1:  PR[91,3] = PR[90,3] + 49.355;
   1:L PR[91] R[100]mm/sec CNT100;
   1:  PR[91,1] = PR[90,1] + 18.409;
   1:  PR[91,2] = PR[90,2] + -16.347;
   1:  PR[91,3] = PR[90,3] + 49.364;
   1:L PR[91] R[100]mm/sec CNT100;
   1:  PR[91,1] = PR[90,1] + 19.270;
   1:  PR[91,2] = PR[90,2] + -15.663;
   1:  PR[91,3] = PR[90,3] + 49.373;
   1:L PR[91] R[100]mm/sec CNT100;
   1:  PR[91,1] = PR[90,1] + 20.094;
   1:  PR[91,2] = PR[90,2] + -14.937;
   1:  PR[91,3] = PR[90,3] + 49.383;
   1:L PR[91] R[100]mm/sec CNT100;
   1:  PR[91,1] = PR[90,1] + 20.878;
   1:  PR[91,2] = PR[90,2] + -14.172;
   1:  PR[91,3] = PR[90,3] + 49.392;
   1:L PR[91] R[100]mm/sec CNT100;
   1:  PR[91,1] = PR[90,1] + 21.621;
   1:  PR[91,2] = PR[90,2] + -13.370;
   1:  PR[91,3] = PR[90,3] + 49.402;
   1:L PR[91] R[100]mm/sec CNT100;
   1:  PR[91,1] = PR[90,1] + 22.320;
   1:  PR[91,2] = PR[90,2] + -12.532;
   1:  PR[91,3] = PR[90,3] + 49.411;
   1:L PR[91] R[100]mm/sec CNT100;
   1:  PR[91,1] = PR[90,1] + 22.975;
   1:  PR[91,2] = PR[90,2] + -11.660;
   1:  PR[91,3] = PR[90,3] + 49.420;
   1:L PR[91] R[100]mm/sec CNT100;
   1:  PR[91,1] = PR[90,1] + 23.583;
   1:  PR[91,2] = PR[90,2] + -10.758;
   1:  PR[91,3] = PR[90,3] + 49.429;
   1:L PR[91] R[100]mm/sec CNT100;
   1:  PR[91,1] = PR[90,1] + 24.143;
   1:  PR[91,2] = PR[90,2] + -9.829;
   1:  PR[91,3] = PR[90,3] + 49.439;
   1:L PR[91] R[100]mm/sec CNT100;
   1:  PR[91,1] = PR[90,1] + 24.654;
   1:  PR[91,2] = PR[90,2] + -8.875;
   1:  PR[91,3] = PR[90,3] + 49.448;
   1:L PR[91] R[100]mm/sec CNT100;
   1:  PR[91,1] = PR[90,1] + 25.115;
   1:  PR[91,2] = PR[90,2] + -7.901;
   1:  PR[91,3] = PR[90,3] + 49.457;
   1:L PR[91] R[100]mm/sec CNT100;
   1:  PR[91,1] = PR[90,1] + 25.524;
   1:  PR[91,2] = PR[90,2] + -6.909;
   1:  PR[91,3] = PR[90,3] + 49.466;
   1:L PR[91] R[100]mm/sec CNT100;
   1:  PR[91,1] = PR[90,1] + 25.880;
   1:  PR[91,2] = PR[90,2] + -5.902;
   1:  PR[91,3] = PR[90,3] + 49.476;
   1:L PR[91] R[100]mm/sec CNT100;
   1:  PR[91,1] = PR[90,1] + 26.182;
   1:  PR[91,2] = PR[90,2] + -4.882;
   1:  PR[91,3] = PR[90,3] + 49.485;
   1:L PR[91] R[100]mm/sec CNT100;
   1:  PR[91,1] = PR[90,1] + 26.431;
   1:  PR[91,2] = PR[90,2] + -3.848;
   1:  PR[91,3] = PR[90,3] + 49.494;
   1:L PR[91] R[100]mm/sec CNT100;
   1:  PR[91,1] = PR[90,1] + 26.625;
   1:  PR[91,2] = PR[90,2] + -2.800;
   1:  PR[91,3] = PR[90,3] + 49.503;
   1:L PR[91] R[100]mm/sec CNT100;
   1:  PR[91,1] = PR[90,1] + 26.764;
   1:  PR[91,2] = PR[90,2] + -1.739;
   1:  PR[91,3] = PR[90,3] + 49.512;
   1:L PR[91] R[100]mm/sec CNT100;
   1:  PR[91,1] = PR[90,1] + 26.847;
   1:  PR[91,2] = PR[90,2] + -0.663;
   1:  PR[91,3] = PR[90,3] + 49.521;
   1:L PR[91] R[100]mm/sec CNT100;
   1:  PR[91,1] = PR[90,1] + 26.875;
   1:  PR[91,2] = PR[90,2] + 0.428;
   1:  PR[91,3] = PR[90,3] + 49.530;
   1:L PR[91] R[100]mm/sec CNT100;
   1:  PR[91,1] = PR[90,1] + 26.847;
   1:  PR[91,2] = PR[90,2] + 1.518;
   1:  PR[91,3] = PR[90,3] + 49.539;
   1:L PR[91] R[100]mm/sec CNT100;
   1:  PR[91,1] = PR[90,1] + 26.764;
   1:  PR[91,2] = PR[90,2] + 2.594;
   1:  PR[91,3] = PR[90,3] + 49.549;
   1:L PR[91] R[100]mm/sec CNT100;
   1:  PR[91,1] = PR[90,1] + 26.625;
   1:  PR[91,2] = PR[90,2] + 3.655;
   1:  PR[91,3] = PR[90,3] + 49.558;
   1:L PR[91] R[100]mm/sec CNT100;
   1:  PR[91,1] = PR[90,1] + 26.431;
   1:  PR[91,2] = PR[90,2] + 4.703;
   1:  PR[91,3] = PR[90,3] + 49.567;
   1:L PR[91] R[100]mm/sec CNT100;
   1:  PR[91,1] = PR[90,1] + 26.183;
   1:  PR[91,2] = PR[90,2] + 5.737;
   1:  PR[91,3] = PR[90,3] + 49.576;
   1:L PR[91] R[100]mm/sec CNT100;
   1:  PR[91,1] = PR[90,1] + 25.880;
   1:  PR[91,2] = PR[90,2] + 6.757;
   1:  PR[91,3] = PR[90,3] + 49.585;
   1:L PR[91] R[100]mm/sec CNT100;
   1:  PR[91,1] = PR[90,1] + 25.524;
   1:  PR[91,2] = PR[90,2] + 7.764;
   1:  PR[91,3] = PR[90,3] + 49.594;
   1:L PR[91] R[100]mm/sec CNT100;
   1:  PR[91,1] = PR[90,1] + 25.115;
   1:  PR[91,2] = PR[90,2] + 8.756;
   1:  PR[91,3] = PR[90,3] + 49.603;
   1:L PR[91] R[100]mm/sec CNT100;
   1:  PR[91,1] = PR[90,1] + 24.655;
   1:  PR[91,2] = PR[90,2] + 9.730;
   1:  PR[91,3] = PR[90,3] + 49.613;
   1:L PR[91] R[100]mm/sec CNT100;
   1:  PR[91,1] = PR[90,1] + 24.144;
   1:  PR[91,2] = PR[90,2] + 10.684;
   1:  PR[91,3] = PR[90,3] + 49.622;
   1:L PR[91] R[100]mm/sec CNT100;
   1:  PR[91,1] = PR[90,1] + 23.583;
   1:  PR[91,2] = PR[90,2] + 11.613;
   1:  PR[91,3] = PR[90,3] + 49.631;
   1:L PR[91] R[100]mm/sec CNT100;
   1:  PR[91,1] = PR[90,1] + 22.975;
   1:  PR[91,2] = PR[90,2] + 12.515;
   1:  PR[91,3] = PR[90,3] + 49.640;
   1:L PR[91] R[100]mm/sec CNT100;
   1:  PR[91,1] = PR[90,1] + 22.321;
   1:  PR[91,2] = PR[90,2] + 13.386;
   1:  PR[91,3] = PR[90,3] + 49.649;
   1:L PR[91] R[100]mm/sec CNT100;
   1:  PR[91,1] = PR[90,1] + 21.621;
   1:  PR[91,2] = PR[90,2] + 14.224;
   1:  PR[91,3] = PR[90,3] + 49.659;
   1:L PR[91] R[100]mm/sec CNT100;
   1:  PR[91,1] = PR[90,1] + 20.879;
   1:  PR[91,2] = PR[90,2] + 15.027;
   1:  PR[91,3] = PR[90,3] + 49.668;
   1:L PR[91] R[100]mm/sec CNT100;
   1:  PR[91,1] = PR[90,1] + 20.095;
   1:  PR[91,2] = PR[90,2] + 15.792;
   1:  PR[91,3] = PR[90,3] + 49.677;
   1:L PR[91] R[100]mm/sec CNT100;
   1:  PR[91,1] = PR[90,1] + 19.271;
   1:  PR[91,2] = PR[90,2] + 16.517;
   1:  PR[91,3] = PR[90,3] + 49.687;
   1:L PR[91] R[100]mm/sec CNT100;
   1:  PR[91,1] = PR[90,1] + 18.410;
   1:  PR[91,2] = PR[90,2] + 17.202;
   1:  PR[91,3] = PR[90,3] + 49.696;
   1:L PR[91] R[100]mm/sec CNT100;
   1:  PR[91,1] = PR[90,1] + 17.513;
   1:  PR[91,2] = PR[90,2] + 17.843;
   1:  PR[91,3] = PR[90,3] + 49.705;
   1:L PR[91] R[100]mm/sec CNT100;
   1:  PR[91,1] = PR[90,1] + 16.583;
   1:  PR[91,2] = PR[90,2] + 18.440;
   1:  PR[91,3] = PR[90,3] + 49.715;
   1:L PR[91] R[100]mm/sec CNT100;
   1:  PR[91,1] = PR[90,1] + 15.623;
   1:  PR[91,2] = PR[90,2] + 18.991;
   1:  PR[91,3] = PR[90,3] + 49.724;
   1:L PR[91] R[100]mm/sec CNT100;
   1:  PR[91,1] = PR[90,1] + 14.634;
   1:  PR[91,2] = PR[90,2] + 19.494;
   1:  PR[91,3] = PR[90,3] + 49.734;
   1:L PR[91] R[100]mm/sec CNT100;
   1:  PR[91,1] = PR[90,1] + 13.619;
   1:  PR[91,2] = PR[90,2] + 19.948;
   1:  PR[91,3] = PR[90,3] + 49.743;
   1:L PR[91] R[100]mm/sec CNT100;
   1:  PR[91,1] = PR[90,1] + 12.582;
   1:  PR[91,2] = PR[90,2] + 20.351;
   1:  PR[91,3] = PR[90,3] + 49.753;
   1:L PR[91] R[100]mm/sec CNT100;
   1:  PR[91,1] = PR[90,1] + 11.524;
   1:  PR[91,2] = PR[90,2] + 20.702;
   1:  PR[91,3] = PR[90,3] + 49.762;
   1:L PR[91] R[100]mm/sec CNT100;
   1:  PR[91,1] = PR[90,1] + 10.448;
   1:  PR[91,2] = PR[90,2] + 21.000;
   1:  PR[91,3] = PR[90,3] + 49.772;
   1:L PR[91] R[100]mm/sec CNT100;
   1:  PR[91,1] = PR[90,1] + 9.357;
   1:  PR[91,2] = PR[90,2] + 21.245;
   1:  PR[91,3] = PR[90,3] + 49.781;
   1:L PR[91] R[100]mm/sec CNT100;
   1:  PR[91,1] = PR[90,1] + 8.254;
   1:  PR[91,2] = PR[90,2] + 21.434;
   1:  PR[91,3] = PR[90,3] + 49.791;
   1:L PR[91] R[100]mm/sec CNT100;
   1:  PR[91,1] = PR[90,1] + 7.142;
   1:  PR[91,2] = PR[90,2] + 21.568;
   1:  PR[91,3] = PR[90,3] + 49.800;
   1:L PR[91] R[100]mm/sec CNT100;
   1:  PR[91,1] = PR[90,1] + 6.024;
   1:  PR[91,2] = PR[90,2] + 21.646;
   1:  PR[91,3] = PR[90,3] + 49.810;
   1:L PR[91] R[100]mm/sec CNT100;
   1:  PR[91,1] = PR[90,1] + 4.902;
   1:  PR[91,2] = PR[90,2] + 21.668;
   1:  PR[91,3] = PR[90,3] + 49.819;
   1:L PR[91] R[100]mm/sec CNT100;
   1:  PR[91,1] = PR[90,1] + 3.781;
   1:  PR[91,2] = PR[90,2] + 21.633;
   1:  PR[91,3] = PR[90,3] + 49.829;
   1:L PR[91] R[100]mm/sec CNT100;
   1:  PR[91,1] = PR[90,1] + 2.662;
   1:  PR[91,2] = PR[90,2] + 21.542;
   1:  PR[91,3] = PR[90,3] + 49.838;
   1:L PR[91] R[100]mm/sec CNT100;
   1:  PR[91,1] = PR[90,1] + 1.536;
   1:  PR[91,2] = PR[90,2] + 21.392;
   1:  PR[91,3] = PR[90,3] + 49.848;
   1:L PR[91] R[100]mm/sec CNT100;
   1:  PR[91,1] = PR[90,1] + 0.234;
   1:  PR[91,2] = PR[90,2] + 21.156;
   1:  PR[91,3] = PR[90,3] + 49.858;
   1:L PR[91] R[100]mm/sec CNT100;
   1:  PR[91,1] = PR[90,1] + -0.250;
   1:  PR[91,2] = PR[90,2] + 21.138;
   1:  PR[91,3] = PR[90,3] + 49.869;
   1:L PR[91] R[100]mm/sec CNT100;
   1:  PR[91,1] = PR[90,1] + -0.703;
   1:  PR[91,2] = PR[90,2] + 21.195;
   1:  PR[91,3] = PR[90,3] + 49.873;
   1:L PR[91] R[100]mm/sec CNT100;
   1:  PR[91,1] = PR[90,1] + -1.784;
   1:  PR[91,2] = PR[90,2] + 21.394;
   1:  PR[91,3] = PR[90,3] + 49.877;
   1:L PR[91] R[100]mm/sec CNT100;
   1:  PR[91,1] = PR[90,1] + -2.899;
   1:  PR[91,2] = PR[90,2] + 21.541;
   1:  PR[91,3] = PR[90,3] + 49.886;
   1:L PR[91] R[100]mm/sec CNT100;
   1:  PR[91,1] = PR[90,1] + -4.018;
   1:  PR[91,2] = PR[90,2] + 21.633;
   1:  PR[91,3] = PR[90,3] + 49.896;
   1:L PR[91] R[100]mm/sec CNT100;
   1:  PR[91,1] = PR[90,1] + -5.139;
   1:  PR[91,2] = PR[90,2] + 21.668;
   1:  PR[91,3] = PR[90,3] + 49.906;
   1:L PR[91] R[100]mm/sec CNT100;
   1:  PR[91,1] = PR[90,1] + -6.261;
   1:  PR[91,2] = PR[90,2] + 21.646;
   1:  PR[91,3] = PR[90,3] + 49.915;
   1:L PR[91] R[100]mm/sec CNT100;
   1:  PR[91,1] = PR[90,1] + -7.379;
   1:  PR[91,2] = PR[90,2] + 21.568;
   1:  PR[91,3] = PR[90,3] + 49.925;
   1:L PR[91] R[100]mm/sec CNT100;
   1:  PR[91,1] = PR[90,1] + -8.491;
   1:  PR[91,2] = PR[90,2] + 21.434;
   1:  PR[91,3] = PR[90,3] + 49.934;
   1:L PR[91] R[100]mm/sec CNT100;
   1:  PR[91,1] = PR[90,1] + -9.594;
   1:  PR[91,2] = PR[90,2] + 21.245;
   1:  PR[91,3] = PR[90,3] + 49.944;
   1:L PR[91] R[100]mm/sec CNT100;
   1:  PR[91,1] = PR[90,1] + -10.685;
   1:  PR[91,2] = PR[90,2] + 21.001;
   1:  PR[91,3] = PR[90,3] + 49.953;
   1:L PR[91] R[100]mm/sec CNT100;
   1:  PR[91,1] = PR[90,1] + -11.761;
   1:  PR[91,2] = PR[90,2] + 20.703;
   1:  PR[91,3] = PR[90,3] + 49.963;
   1:L PR[91] R[100]mm/sec CNT100;
   1:  PR[91,1] = PR[90,1] + -12.819;
   1:  PR[91,2] = PR[90,2] + 20.352;
   1:  PR[91,3] = PR[90,3] + 49.972;
   1:L PR[91] R[100]mm/sec CNT100;
   1:  PR[91,1] = PR[90,1] + -13.857;
   1:  PR[91,2] = PR[90,2] + 19.949;
   1:  PR[91,3] = PR[90,3] + 49.982;
   1:L PR[91] R[100]mm/sec CNT100;
   1:  PR[91,1] = PR[90,1] + -14.871;
   1:  PR[91,2] = PR[90,2] + 19.494;
   1:  PR[91,3] = PR[90,3] + 49.991;
   1:L PR[91] R[100]mm/sec CNT100;
   1:  PR[91,1] = PR[90,1] + -15.860;
   1:  PR[91,2] = PR[90,2] + 18.991;
   1:  PR[91,3] = PR[90,3] + 50.001;
   1:L PR[91] R[100]mm/sec CNT100;
   1:  PR[91,1] = PR[90,1] + -16.821;
   1:  PR[91,2] = PR[90,2] + 18.440;
   1:  PR[91,3] = PR[90,3] + 50.010;
   1:L PR[91] R[100]mm/sec CNT100;
   1:  PR[91,1] = PR[90,1] + -17.751;
   1:  PR[91,2] = PR[90,2] + 17.843;
   1:  PR[91,3] = PR[90,3] + 50.020;
   1:L PR[91] R[100]mm/sec CNT100;
   1:  PR[91,1] = PR[90,1] + -18.647;
   1:  PR[91,2] = PR[90,2] + 17.201;
   1:  PR[91,3] = PR[90,3] + 50.029;
   1:L PR[91] R[100]mm/sec CNT100;
   1:  PR[91,1] = PR[90,1] + -19.509;
   1:  PR[91,2] = PR[90,2] + 16.517;
   1:  PR[91,3] = PR[90,3] + 50.039;
   1:L PR[91] R[100]mm/sec CNT100;
   1:  PR[91,1] = PR[90,1] + -20.333;
   1:  PR[91,2] = PR[90,2] + 15.792;
   1:  PR[91,3] = PR[90,3] + 50.048;
   1:L PR[91] R[100]mm/sec CNT100;
   1:  PR[91,1] = PR[90,1] + -21.117;
   1:  PR[91,2] = PR[90,2] + 15.027;
   1:  PR[91,3] = PR[90,3] + 50.057;
   1:L PR[91] R[100]mm/sec CNT100;
   1:  PR[91,1] = PR[90,1] + -21.860;
   1:  PR[91,2] = PR[90,2] + 14.226;
   1:  PR[91,3] = PR[90,3] + 50.067;
   1:L PR[91] R[100]mm/sec CNT100;
   1:  PR[91,1] = PR[90,1] + -22.559;
   1:  PR[91,2] = PR[90,2] + 13.389;
   1:  PR[91,3] = PR[90,3] + 50.076;
   1:L PR[91] R[100]mm/sec CNT100;
   1:  PR[91,1] = PR[90,1] + -23.214;
   1:  PR[91,2] = PR[90,2] + 12.518;
   1:  PR[91,3] = PR[90,3] + 50.085;
   1:L PR[91] R[100]mm/sec CNT100;
   1:  PR[91,1] = PR[90,1] + -23.822;
   1:  PR[91,2] = PR[90,2] + 11.617;
   1:  PR[91,3] = PR[90,3] + 50.094;
   1:L PR[91] R[100]mm/sec CNT100;
   1:  PR[91,1] = PR[90,1] + -24.382;
   1:  PR[91,2] = PR[90,2] + 10.687;
   1:  PR[91,3] = PR[90,3] + 50.104;
   1:L PR[91] R[100]mm/sec CNT100;
   1:  PR[91,1] = PR[90,1] + -24.893;
   1:  PR[91,2] = PR[90,2] + 9.732;
   1:  PR[91,3] = PR[90,3] + 50.113;
   1:L PR[91] R[100]mm/sec CNT100;
   1:  PR[91,1] = PR[90,1] + -25.353;
   1:  PR[91,2] = PR[90,2] + 8.756;
   1:  PR[91,3] = PR[90,3] + 50.122;
   1:L PR[91] R[100]mm/sec CNT100;
   1:  PR[91,1] = PR[90,1] + -25.762;
   1:  PR[91,2] = PR[90,2] + 7.761;
   1:  PR[91,3] = PR[90,3] + 50.131;
   1:L PR[91] R[100]mm/sec CNT100;
   1:  PR[91,1] = PR[90,1] + -26.118;
   1:  PR[91,2] = PR[90,2] + 6.752;
   1:  PR[91,3] = PR[90,3] + 50.141;
   1:L PR[91] R[100]mm/sec CNT100;
   1:  PR[91,1] = PR[90,1] + -26.421;
   1:  PR[91,2] = PR[90,2] + 5.731;
   1:  PR[91,3] = PR[90,3] + 50.150;
   1:L PR[91] R[100]mm/sec CNT100;
   1:  PR[91,1] = PR[90,1] + -26.669;
   1:  PR[91,2] = PR[90,2] + 4.697;
   1:  PR[91,3] = PR[90,3] + 50.159;
   1:L PR[91] R[100]mm/sec CNT100;
   1:  PR[91,1] = PR[90,1] + -26.863;
   1:  PR[91,2] = PR[90,2] + 3.651;
   1:  PR[91,3] = PR[90,3] + 50.168;
   1:L PR[91] R[100]mm/sec CNT100;
   1:  PR[91,1] = PR[90,1] + -27.002;
   1:  PR[91,2] = PR[90,2] + 2.592;
   1:  PR[91,3] = PR[90,3] + 50.177;
   1:L PR[91] R[100]mm/sec CNT100;
   1:  PR[91,1] = PR[90,1] + -27.086;
   1:  PR[91,2] = PR[90,2] + 1.517;
   1:  PR[91,3] = PR[90,3] + 50.186;
   1:L PR[91] R[100]mm/sec CNT100;
   1:  PR[91,1] = PR[90,1] + -27.114;
   1:  PR[91,2] = PR[90,2] + 0.428;
   1:  PR[91,3] = PR[90,3] + 50.195;
   1:L PR[91] R[100]mm/sec CNT100;
   1:  PR[91,1] = PR[90,1] + -27.086;
   1:  PR[91,2] = PR[90,2] + -0.662;
   1:  PR[91,3] = PR[90,3] + 50.204;
   1:L PR[91] R[100]mm/sec CNT100;
   1:  PR[91,1] = PR[90,1] + -27.002;
   1:  PR[91,2] = PR[90,2] + -1.737;
   1:  PR[91,3] = PR[90,3] + 50.214;
   1:L PR[91] R[100]mm/sec CNT100;
   1:  PR[91,1] = PR[90,1] + -26.863;
   1:  PR[91,2] = PR[90,2] + -2.796;
   1:  PR[91,3] = PR[90,3] + 50.223;
   1:L PR[91] R[100]mm/sec CNT100;
   1:  PR[91,1] = PR[90,1] + -26.669;
   1:  PR[91,2] = PR[90,2] + -3.842;
   1:  PR[91,3] = PR[90,3] + 50.232;
   1:L PR[91] R[100]mm/sec CNT100;
   1:  PR[91,1] = PR[90,1] + -26.421;
   1:  PR[91,2] = PR[90,2] + -4.876;
   1:  PR[91,3] = PR[90,3] + 50.241;
   1:L PR[91] R[100]mm/sec CNT100;
   1:  PR[91,1] = PR[90,1] + -26.118;
   1:  PR[91,2] = PR[90,2] + -5.898;
   1:  PR[91,3] = PR[90,3] + 50.250;
   1:L PR[91] R[100]mm/sec CNT100;
   1:  PR[91,1] = PR[90,1] + -25.762;
   1:  PR[91,2] = PR[90,2] + -6.907;
   1:  PR[91,3] = PR[90,3] + 50.259;
   1:L PR[91] R[100]mm/sec CNT100;
   1:  PR[91,1] = PR[90,1] + -25.353;
   1:  PR[91,2] = PR[90,2] + -7.901;
   1:  PR[91,3] = PR[90,3] + 50.268;
   1:L PR[91] R[100]mm/sec CNT100;
   1:  PR[91,1] = PR[90,1] + -24.892;
   1:  PR[91,2] = PR[90,2] + -8.878;
   1:  PR[91,3] = PR[90,3] + 50.278;
   1:L PR[91] R[100]mm/sec CNT100;
   1:  PR[91,1] = PR[90,1] + -24.382;
   1:  PR[91,2] = PR[90,2] + -9.832;
   1:  PR[91,3] = PR[90,3] + 50.287;
   1:L PR[91] R[100]mm/sec CNT100;
   1:  PR[91,1] = PR[90,1] + -23.821;
   1:  PR[91,2] = PR[90,2] + -10.762;
   1:  PR[91,3] = PR[90,3] + 50.296;
   1:L PR[91] R[100]mm/sec CNT100;
   1:  PR[91,1] = PR[90,1] + -23.213;
   1:  PR[91,2] = PR[90,2] + -11.664;
   1:  PR[91,3] = PR[90,3] + 50.305;
   1:L PR[91] R[100]mm/sec CNT100;
   1:  PR[91,1] = PR[90,1] + -22.559;
   1:  PR[91,2] = PR[90,2] + -12.534;
   1:  PR[91,3] = PR[90,3] + 50.315;
   1:L PR[91] R[100]mm/sec CNT100;
   1:  PR[91,1] = PR[90,1] + -21.859;
   1:  PR[91,2] = PR[90,2] + -13.371;
   1:  PR[91,3] = PR[90,3] + 50.324;
   1:L PR[91] R[100]mm/sec CNT100;
   1:  PR[91,1] = PR[90,1] + -21.116;
   1:  PR[91,2] = PR[90,2] + -14.173;
   1:  PR[91,3] = PR[90,3] + 50.333;
   1:L PR[91] R[100]mm/sec CNT100;
   1:  PR[91,1] = PR[90,1] + -20.332;
   1:  PR[91,2] = PR[90,2] + -14.937;
   1:  PR[91,3] = PR[90,3] + 50.342;
   1:L PR[91] R[100]mm/sec CNT100;
   1:  PR[91,1] = PR[90,1] + -19.508;
   1:  PR[91,2] = PR[90,2] + -15.662;
   1:  PR[91,3] = PR[90,3] + 50.352;
   1:L PR[91] R[100]mm/sec CNT100;
   1:  PR[91,1] = PR[90,1] + -18.646;
   1:  PR[91,2] = PR[90,2] + -16.347;
   1:  PR[91,3] = PR[90,3] + 50.361;
   1:L PR[91] R[100]mm/sec CNT100;
   1:  PR[91,1] = PR[90,1] + -17.750;
   1:  PR[91,2] = PR[90,2] + -16.988;
   1:  PR[91,3] = PR[90,3] + 50.370;
   1:L PR[91] R[100]mm/sec CNT100;
   1:  PR[91,1] = PR[90,1] + -16.820;
   1:  PR[91,2] = PR[90,2] + -17.586;
   1:  PR[91,3] = PR[90,3] + 50.380;
   1:L PR[91] R[100]mm/sec CNT100;
   1:  PR[91,1] = PR[90,1] + -15.859;
   1:  PR[91,2] = PR[90,2] + -18.137;
   1:  PR[91,3] = PR[90,3] + 50.389;
   1:L PR[91] R[100]mm/sec CNT100;
   1:  PR[91,1] = PR[90,1] + -14.870;
   1:  PR[91,2] = PR[90,2] + -18.640;
   1:  PR[91,3] = PR[90,3] + 50.399;
   1:L PR[91] R[100]mm/sec CNT100;
   1:  PR[91,1] = PR[90,1] + -13.855;
   1:  PR[91,2] = PR[90,2] + -19.094;
   1:  PR[91,3] = PR[90,3] + 50.408;
   1:L PR[91] R[100]mm/sec CNT100;
   1:  PR[91,1] = PR[90,1] + -12.818;
   1:  PR[91,2] = PR[90,2] + -19.497;
   1:  PR[91,3] = PR[90,3] + 50.418;
   1:L PR[91] R[100]mm/sec CNT100;
   1:  PR[91,1] = PR[90,1] + -11.759;
   1:  PR[91,2] = PR[90,2] + -19.848;
   1:  PR[91,3] = PR[90,3] + 50.427;
   1:L PR[91] R[100]mm/sec CNT100;
   1:  PR[91,1] = PR[90,1] + -10.683;
   1:  PR[91,2] = PR[90,2] + -20.146;
   1:  PR[91,3] = PR[90,3] + 50.437;
   1:L PR[91] R[100]mm/sec CNT100;
   1:  PR[91,1] = PR[90,1] + -9.592;
   1:  PR[91,2] = PR[90,2] + -20.390;
   1:  PR[91,3] = PR[90,3] + 50.446;
   1:L PR[91] R[100]mm/sec CNT100;
   1:  PR[91,1] = PR[90,1] + -8.489;
   1:  PR[91,2] = PR[90,2] + -20.580;
   1:  PR[91,3] = PR[90,3] + 50.456;
   1:L PR[91] R[100]mm/sec CNT100;
   1:  PR[91,1] = PR[90,1] + -7.377;
   1:  PR[91,2] = PR[90,2] + -20.713;
   1:  PR[91,3] = PR[90,3] + 50.465;
   1:L PR[91] R[100]mm/sec CNT100;
   1:  PR[91,1] = PR[90,1] + -6.259;
   1:  PR[91,2] = PR[90,2] + -20.791;
   1:  PR[91,3] = PR[90,3] + 50.475;
   1:L PR[91] R[100]mm/sec CNT100;
   1:  PR[91,1] = PR[90,1] + -5.137;
   1:  PR[91,2] = PR[90,2] + -20.813;
   1:  PR[91,3] = PR[90,3] + 50.484;
   1:L PR[91] R[100]mm/sec CNT100;
   1:  PR[91,1] = PR[90,1] + -4.016;
   1:  PR[91,2] = PR[90,2] + -20.778;
   1:  PR[91,3] = PR[90,3] + 50.494;
   1:L PR[91] R[100]mm/sec CNT100;
   1:  PR[91,1] = PR[90,1] + -2.897;
   1:  PR[91,2] = PR[90,2] + -20.686;
   1:  PR[91,3] = PR[90,3] + 50.503;
   1:L PR[91] R[100]mm/sec CNT100;
   1:  PR[91,1] = PR[90,1] + -1.774;
   1:  PR[91,2] = PR[90,2] + -20.537;
   1:  PR[91,3] = PR[90,3] + 50.513;
   1:L PR[91] R[100]mm/sec CNT100;
   1:  PR[91,1] = PR[90,1] + -0.703;
   1:  PR[91,2] = PR[90,2] + -20.340;
   1:  PR[91,3] = PR[90,3] + 50.523;
   1:L PR[91] R[100]mm/sec CNT100;
   1:  PR[91,1] = PR[90,1] + -0.250;
   1:  PR[91,2] = PR[90,2] + -20.282;
   1:  PR[91,3] = PR[90,3] + 50.532;
   1:L PR[91] R[100]mm/sec CNT100;
   1:  PR[91,1] = PR[90,1] + 0.233;
   1:  PR[91,2] = PR[90,2] + -20.301;
   1:  PR[91,3] = PR[90,3] + 50.536;
   1:L PR[91] R[100]mm/sec CNT100;
   1:  PR[91] = PR[90];
   1:  PR[91,1] = PR[90,1] + 0.974;
   1:  PR[91,2] = PR[90,2] + -20.794;
   1:  PR[91,3] = PR[90,3] + 51.870;
   1:L PR[91] R[100]mm/sec CNT100;
   1:  PR[91,1] = PR[90,1] + 2.105;
   1:  PR[91,2] = PR[90,2] + -20.946;
   1:  PR[91,3] = PR[90,3] + 50.546;
   1:L PR[91] R[100]mm/sec CNT100;
   1:  PR[91,1] = PR[90,1] + 3.237;
   1:  PR[91,2] = PR[90,2] + -21.039;
   1:  PR[91,3] = PR[90,3] + 50.556;
   1:L PR[91] R[100]mm/sec CNT100;
   1:  PR[91,1] = PR[90,1] + 4.371;
   1:  PR[91,2] = PR[90,2] + -21.076;
   1:  PR[91,3] = PR[90,3] + 50.565;
   1:L PR[91] R[100]mm/sec CNT100;
   1:  PR[91,1] = PR[90,1] + 5.506;
   1:  PR[91,2] = PR[90,2] + -21.055;
   1:  PR[91,3] = PR[90,3] + 50.575;
   1:L PR[91] R[100]mm/sec CNT100;
   1:  PR[91,1] = PR[90,1] + 5.901;
   1:  PR[91,2] = PR[90,2] + -21.028;
   1:  PR[91,3] = PR[90,3] + 50.585;
   1:L PR[91] R[100]mm/sec CNT100;
   1:  PR[91,1] = PR[90,1] + 6.636;
   1:  PR[91,2] = PR[90,2] + -20.976;
   1:  PR[91,3] = PR[90,3] + 50.588;
   1:L PR[91] R[100]mm/sec CNT100;
   1:  PR[91,1] = PR[90,1] + 7.761;
   1:  PR[91,2] = PR[90,2] + -20.841;
   1:  PR[91,3] = PR[90,3] + 50.595;
   1:L PR[91] R[100]mm/sec CNT100;
   1:  PR[91,1] = PR[90,1] + 8.876;
   1:  PR[91,2] = PR[90,2] + -20.650;
   1:  PR[91,3] = PR[90,3] + 50.604;
   1:L PR[91] R[100]mm/sec CNT100;
   1:  PR[91,1] = PR[90,1] + 9.980;
   1:  PR[91,2] = PR[90,2] + -20.402;
   1:  PR[91,3] = PR[90,3] + 50.614;
   1:L PR[91] R[100]mm/sec CNT100;
   1:  PR[91,1] = PR[90,1] + 11.067;
   1:  PR[91,2] = PR[90,2] + -20.100;
   1:  PR[91,3] = PR[90,3] + 50.624;
   1:L PR[91] R[100]mm/sec CNT100;
   1:  PR[91,1] = PR[90,1] + 12.138;
   1:  PR[91,2] = PR[90,2] + -19.744;
   1:  PR[91,3] = PR[90,3] + 50.633;
   1:L PR[91] R[100]mm/sec CNT100;
   1:  PR[91,1] = PR[90,1] + 13.186;
   1:  PR[91,2] = PR[90,2] + -19.336;
   1:  PR[91,3] = PR[90,3] + 50.643;
   1:L PR[91] R[100]mm/sec CNT100;
   1:  PR[91,1] = PR[90,1] + 14.212;
   1:  PR[91,2] = PR[90,2] + -18.876;
   1:  PR[91,3] = PR[90,3] + 50.653;
   1:L PR[91] R[100]mm/sec CNT100;
   1:  PR[91,1] = PR[90,1] + 15.212;
   1:  PR[91,2] = PR[90,2] + -18.367;
   1:  PR[91,3] = PR[90,3] + 50.662;
   1:L PR[91] R[100]mm/sec CNT100;
   1:  PR[91,1] = PR[90,1] + 16.182;
   1:  PR[91,2] = PR[90,2] + -17.809;
   1:  PR[91,3] = PR[90,3] + 50.672;
   1:L PR[91] R[100]mm/sec CNT100;
   1:  PR[91,1] = PR[90,1] + 17.123;
   1:  PR[91,2] = PR[90,2] + -17.203;
   1:  PR[91,3] = PR[90,3] + 50.681;
   1:L PR[91] R[100]mm/sec CNT100;
   1:  PR[91,1] = PR[90,1] + 18.028;
   1:  PR[91,2] = PR[90,2] + -16.555;
   1:  PR[91,3] = PR[90,3] + 50.691;
   1:L PR[91] R[100]mm/sec CNT100;
   1:  PR[91,1] = PR[90,1] + 18.898;
   1:  PR[91,2] = PR[90,2] + -15.863;
   1:  PR[91,3] = PR[90,3] + 50.700;
   1:L PR[91] R[100]mm/sec CNT100;
   1:  PR[91,1] = PR[90,1] + 19.730;
   1:  PR[91,2] = PR[90,2] + -15.129;
   1:  PR[91,3] = PR[90,3] + 50.710;
   1:L PR[91] R[100]mm/sec CNT100;
   1:  PR[91,1] = PR[90,1] + 20.522;
   1:  PR[91,2] = PR[90,2] + -14.356;
   1:  PR[91,3] = PR[90,3] + 50.719;
   1:L PR[91] R[100]mm/sec CNT100;
   1:  PR[91,1] = PR[90,1] + 21.273;
   1:  PR[91,2] = PR[90,2] + -13.544;
   1:  PR[91,3] = PR[90,3] + 50.729;
   1:L PR[91] R[100]mm/sec CNT100;
   1:  PR[91,1] = PR[90,1] + 21.980;
   1:  PR[91,2] = PR[90,2] + -12.696;
